SPLINE
SPL {X  -126.527, Y  +769.417, Z    +0.000, E1  +405.012, E3 -205837.853}
SPL {X  -145.458, Y  +738.125, Z    +0.000, E1  +396.959, E3 -205873.935}
SPL {X  -156.272, Y  +705.789, Z    +0.000, E1  +383.396, E3 -205888.344}
SPL {X  -159.413, Y  +685.076, Z    +0.000, E1  +371.341, E3 -205892.483}
SPL {X  -159.901, Y  +676.826, Z    +0.000, E1  +365.664, E3 -205893.315}
SPL {X  -159.990, Y  +671.106, Z    +0.000, E1  +361.459, E3 -205893.577}
SPL {X  -159.990, Y  +668.525, Z    +0.000, E1  +359.125, E3 -205893.622}
SPL {X  -159.990, Y  +664.817, Z    +0.000, E1  +353.836, E3 -205893.763}
SPL {X  -159.990, Y  +661.286, Z    +0.000, E1  +348.294, E3 -205894.024}
SPL {X  -159.990, Y  +654.198, Z    +0.000, E1  +336.753, E3 -205894.936}
SPL {X  -159.990, Y  +643.777, Z    +0.000, E1  +322.140, E3 -205897.101}
SPL {X  -159.990, Y  +634.027, Z    +0.000, E1  +313.116, E3 -205900.013}
SPL {X  -159.990, Y  +589.014, Z    +0.000, E1  +298.500, E3 -205920.064}
SPL {X  -159.990, Y  +484.717, Z    +0.000, E1  +295.169, E3 -205998.247}
SPL {X  -159.990, Y  +469.712, Z    +0.000, E1  +295.152, E3 -206013.185}
SPL {X  -159.990, Y  +456.089, Z    +0.000, E1  +295.174, E3 -206026.800}
SPL {X  -159.990, Y  +443.816, Z    +0.000, E1  +295.158, E3 -206039.000}
SPL {X  -159.990, Y  +405.035, Z    +0.000, E1  +292.209, E3 -206051.271}
SPL {X  -159.990, Y  +395.217, Z    +0.000, E1  +293.078, E3 -206067.380}
SPL {X  -159.990, Y  +385.177, Z    +0.000, E1  +294.011, E3 -206084.069}
SPL {X  -159.935, Y  +378.300, Z    +0.000, E1  +295.100, E3 -206099.278}
SPL {X  -159.533, Y  +370.414, Z    +0.000, E1  +296.253, E3 -206116.187}
SPL {X  -158.431, Y  +360.219, Z    +0.000, E1  +296.670, E3 -206129.704}
SPL {X  -157.299, Y  +353.279, Z    +0.000, E1  +296.835, E3 -206138.201}
SPL {X  -155.242, Y  +343.812, Z    +0.000, E1  +297.102, E3 -206150.249}
SPL {X  -151.999, Y  +332.569, Z    +0.000, E1  +297.592, E3 -206165.407}
SPL {X  -148.909, Y  +323.994, Z    +0.000, E1  +298.107, E3 -206177.581}
SPL {X  -146.667, Y  +318.581, Z    +0.000, E1  +298.485, E3 -206185.501}
SPL {X  -144.416, Y  +313.647, Z    +0.000, E1  +298.845, E3 -206192.837}
SPL {X  -141.484, Y  +307.808, Z    +0.000, E1  +299.342, E3 -206201.730}
SPL {X  -139.055, Y  +303.377, Z    +0.000, E1  +299.788, E3 -206208.642}
SPL {X  -136.464, Y  +298.988, Z    +0.000, E1  +300.231, E3 -206215.517}
SPL {X  -133.486, Y  +294.305, Z    +0.000, E1  +300.785, E3 -206222.979}
SPL {X  -111.198, Y  +267.470, Z    +0.000, E1  +308.990, E3 -206323.999}
ENDSPLINE

SPLINE
SPL {X  -136.508, Y  +299.059, Z    +0.000, E1  +318.212, E3 -206434.935}
SPL {X  -153.176, Y  +336.305, Z    +0.000, E1  +330.872, E3 -206461.500}
SPL {X  -158.263, Y  +359.056, Z    +0.000, E1  +342.551, E3 -206468.175}
SPL {X  -159.616, Y  +371.564, Z    +0.000, E1  +350.434, E3 -206470.080}
SPL {X  -159.983, Y  +381.031, Z    +0.000, E1  +357.053, E3 -206470.771}
SPL {X  -159.990, Y  +384.524, Z    +0.000, E1  +359.995, E3 -206470.859}
SPL {X  -159.990, Y  +386.890, Z    +0.000, E1  +362.742, E3 -206470.915}
SPL {X  -159.990, Y  +392.248, Z    +0.000, E1  +370.895, E3 -206471.242}
SPL {X  -159.990, Y  +398.030, Z    +0.000, E1  +380.706, E3 -206471.894}
SPL {X  -159.990, Y  +404.858, Z    +0.000, E1  +391.125, E3 -206473.138}
SPL {X  -159.990, Y  +416.328, Z    +0.000, E1  +404.105, E3 -206476.075}
SPL {X  -159.990, Y  +459.824, Z    +0.000, E1  +420.326, E3 -206495.997}
SPL {X  -159.990, Y  +561.459, Z    +0.000, E1  +423.923, E3 -206574.863}
SPL {X  -159.990, Y  +574.787, Z    +0.000, E1  +423.950, E3 -206588.660}
SPL {X  -159.990, Y  +590.041, Z    +0.000, E1  +423.939, E3 -206604.520}
SPL {X  -159.990, Y  +601.352, Z    +0.000, E1  +423.918, E3 -206616.306}
SPL {X  -159.990, Y  +610.973, Z    +0.000, E1  +423.927, E3 -206626.274}
SPL {X  -159.990, Y  +624.756, Z    +0.000, E1  +423.949, E3 -206640.552}
SPL {X  -159.990, Y  +640.674, Z    +0.000, E1  +423.943, E3 -206657.089}
SPL {X  -159.990, Y  +652.355, Z    +0.000, E1  +423.915, E3 -206669.287}
SPL {X  -159.990, Y  +661.195, Z    +0.000, E1  +423.915, E3 -206678.486}
SPL {X  -159.965, Y  +674.349, Z    +0.000, E1  +423.939, E3 -206692.123}
SPL {X  -159.404, Y  +685.179, Z    +0.000, E1  +423.831, E3 -206704.002}
SPL {X  -158.535, Y  +693.032, Z    +0.000, E1  +423.713, E3 -206713.051}
SPL {X  -156.949, Y  +702.544, Z    +0.000, E1  +423.501, E3 -206724.557}
SPL {X  -154.903, Y  +711.525, Z    +0.000, E1  +423.186, E3 -206736.028}
SPL {X  -153.138, Y  +717.820, Z    +0.000, E1  +422.909, E3 -206744.382}
SPL {X  -151.229, Y  +723.716, Z    +0.000, E1  +422.630, E3 -206752.392}
SPL {X  -148.422, Y  +731.231, Z    +0.000, E1  +422.207, E3 -206762.950}
SPL {X  -145.802, Y  +737.367, Z    +0.000, E1  +421.758, E3 -206771.902}
SPL {X  -143.476, Y  +742.291, Z    +0.000, E1  +421.379, E3 -206779.203}
SPL {X  -141.015, Y  +747.074, Z    +0.000, E1  +420.958, E3 -206786.459}
SPL {X  -138.539, Y  +751.523, Z    +0.000, E1  +420.526, E3 -206793.294}
SPL {X  -136.299, Y  +755.281, Z    +0.000, E1  +420.128, E3 -206799.155}
SPL {X  -133.306, Y  +759.967, Z    +0.000, E1  +419.584, E3 -206806.550}
SPL {X  -112.019, Y  +785.730, Z    +0.000, E1  +410.795, E3 -206909.290}
ENDSPLINE

SPLINE
SPL {X  -138.335, Y  +751.876, Z    +0.000, E1  +401.001, E3 -207023.589}
SPL {X  -153.384, Y  +716.997, Z    +0.000, E1  +388.774, E3 -207045.960}
SPL {X  -158.303, Y  +694.673, Z    +0.000, E1  +377.238, E3 -207052.272}
SPL {X  -159.604, Y  +682.609, Z    +0.000, E1  +369.664, E3 -207054.082}
SPL {X  -159.964, Y  +674.389, Z    +0.000, E1  +363.956, E3 -207054.744}
SPL {X  -159.990, Y  +669.409, Z    +0.000, E1  +360.015, E3 -207054.897}
SPL {X  -159.990, Y  +666.004, Z    +0.000, E1  +355.742, E3 -207054.998}
SPL {X  -159.990, Y  +661.286, Z    +0.000, E1  +348.294, E3 -207055.315}
SPL {X  -159.990, Y  +656.470, Z    +0.000, E1  +340.220, E3 -207055.852}
SPL {X  -159.990, Y  +651.555, Z    +0.000, E1  +332.416, E3 -207056.660}
SPL {X  -159.990, Y  +640.109, Z    +0.000, E1  +318.471, E3 -207059.489}
SPL {X  -159.990, Y  +589.014, Z    +0.000, E1  +298.500, E3 -207081.355}
SPL {X  -159.990, Y  +484.717, Z    +0.000, E1  +295.169, E3 -207159.538}
SPL {X  -159.990, Y  +474.300, Z    +0.000, E1  +295.184, E3 -207169.966}
SPL {X  -159.990, Y  +460.248, Z    +0.000, E1  +295.138, E3 -207183.876}
SPL {X  -159.990, Y  +443.816, Z    +0.000, E1  +295.158, E3 -207200.291}
SPL {X  -159.990, Y  +405.035, Z    +0.000, E1  +292.209, E3 -207212.562}
SPL {X  -159.990, Y  +397.824, Z    +0.000, E1  +292.709, E3 -207222.924}
SPL {X  -159.990, Y  +393.786, Z    +0.000, E1  +293.391, E3 -207232.243}
SPL {X  -159.990, Y  +387.038, Z    +0.000, E1  +293.844, E3 -207242.098}
SPL {X  -159.983, Y  +380.995, Z    +0.000, E1  +294.559, E3 -207253.667}
SPL {X  -159.898, Y  +377.064, Z    +0.000, E1  +295.481, E3 -207264.481}
SPL {X  -159.533, Y  +370.414, Z    +0.000, E1  +296.253, E3 -207277.478}
SPL {X  -158.431, Y  +360.219, Z    +0.000, E1  +296.670, E3 -207290.995}
SPL {X  -156.653, Y  +349.995, Z    +0.000, E1  +296.892, E3 -207303.563}
SPL {X  -153.792, Y  +338.401, Z    +0.000, E1  +297.323, E3 -207318.732}
SPL {X  -151.244, Y  +330.327, Z    +0.000, E1  +297.748, E3 -207329.885}
SPL {X  -148.909, Y  +323.994, Z    +0.000, E1  +298.107, E3 -207338.871}
SPL {X  -146.667, Y  +318.581, Z    +0.000, E1  +298.485, E3 -207346.791}
SPL {X  -144.416, Y  +313.647, Z    +0.000, E1  +298.845, E3 -207354.127}
SPL {X  -141.484, Y  +307.808, Z    +0.000, E1  +299.342, E3 -207363.020}
SPL {X  -139.055, Y  +303.377, Z    +0.000, E1  +299.788, E3 -207369.933}
SPL {X  -136.464, Y  +298.988, Z    +0.000, E1  +300.231, E3 -207376.807}
SPL {X  -133.486, Y  +294.305, Z    +0.000, E1  +300.785, E3 -207384.269}
SPL {X  -111.268, Y  +267.538, Z    +0.000, E1  +309.436, E3 -207492.168}
ENDSPLINE

SPLINE
SPL {X  -140.331, Y  +305.662, Z    +0.000, E1  +319.927, E3 -207604.236}
SPL {X  -153.176, Y  +336.305, Z    +0.000, E1  +330.872, E3 -207622.791}
SPL {X  -158.263, Y  +359.056, Z    +0.000, E1  +342.551, E3 -207629.465}
SPL {X  -159.616, Y  +371.564, Z    +0.000, E1  +350.434, E3 -207631.370}
SPL {X  -159.983, Y  +381.031, Z    +0.000, E1  +357.053, E3 -207632.061}
SPL {X  -159.990, Y  +384.524, Z    +0.000, E1  +359.995, E3 -207632.149}
SPL {X  -159.990, Y  +386.890, Z    +0.000, E1  +362.742, E3 -207632.205}
SPL {X  -159.990, Y  +392.248, Z    +0.000, E1  +370.895, E3 -207632.533}
SPL {X  -159.990, Y  +398.030, Z    +0.000, E1  +380.706, E3 -207633.184}
SPL {X  -159.990, Y  +404.858, Z    +0.000, E1  +391.125, E3 -207634.428}
SPL {X  -159.990, Y  +416.328, Z    +0.000, E1  +404.105, E3 -207637.365}
SPL {X  -159.990, Y  +459.824, Z    +0.000, E1  +420.326, E3 -207657.287}
SPL {X  -159.990, Y  +565.974, Z    +0.000, E1  +423.959, E3 -207740.776}
SPL {X  -159.990, Y  +582.903, Z    +0.000, E1  +423.951, E3 -207758.373}
SPL {X  -159.990, Y  +598.374, Z    +0.000, E1  +423.941, E3 -207774.459}
SPL {X  -159.990, Y  +614.998, Z    +0.000, E1  +423.962, E3 -207791.681}
SPL {X  -159.990, Y  +632.576, Z    +0.000, E1  +423.953, E3 -207809.947}
SPL {X  -159.990, Y  +648.849, Z    +0.000, E1  +423.945, E3 -207826.876}
SPL {X  -159.990, Y  +665.748, Z    +0.000, E1  +423.953, E3 -207844.431}
SPL {X  -159.643, Y  +682.032, Z    +0.000, E1  +423.894, E3 -207861.725}
SPL {X  -158.070, Y  +696.212, Z    +0.000, E1  +423.682, E3 -207878.063}
SPL {X  -155.481, Y  +709.215, Z    +0.000, E1  +423.310, E3 -207894.254}
SPL {X  -153.138, Y  +717.820, Z    +0.000, E1  +422.909, E3 -207905.672}
SPL {X  -151.229, Y  +723.716, Z    +0.000, E1  +422.630, E3 -207913.682}
SPL {X  -149.219, Y  +729.211, Z    +0.000, E1  +422.307, E3 -207921.390}
SPL {X  -146.537, Y  +735.716, Z    +0.000, E1  +421.906, E3 -207930.733}
SPL {X  -143.476, Y  +742.291, Z    +0.000, E1  +421.379, E3 -207940.493}
SPL {X  -141.015, Y  +747.074, Z    +0.000, E1  +420.958, E3 -207947.750}
SPL {X  -137.271, Y  +753.679, Z    +0.000, E1  +420.346, E3 -207957.888}
SPL {X  -133.306, Y  +759.967, Z    +0.000, E1  +419.584, E3 -207967.840}
SPL {X  -112.019, Y  +785.730, Z    +0.000, E1  +410.795, E3 -208070.581}
ENDSPLINE

SPLINE
SPL {X  -138.335, Y  +751.876, Z    +0.000, E1  +401.001, E3 -208184.879}
SPL {X  -150.285, Y  +726.376, Z    +0.000, E1  +392.667, E3 -208203.288}
SPL {X  -156.272, Y  +705.789, Z    +0.000, E1  +383.396, E3 -208210.925}
SPL {X  -159.413, Y  +685.076, Z    +0.000, E1  +371.341, E3 -208215.063}
SPL {X  -159.964, Y  +674.389, Z    +0.000, E1  +363.956, E3 -208216.034}
SPL {X  -159.990, Y  +670.214, Z    +0.000, E1  +360.653, E3 -208216.180}
SPL {X  -159.990, Y  +669.154, Z    +0.000, E1  +359.694, E3 -208216.189}
SPL {X  -159.990, Y  +666.004, Z    +0.000, E1  +355.742, E3 -208216.289}
SPL {X  -159.990, Y  +661.286, Z    +0.000, E1  +348.294, E3 -208216.605}
SPL {X  -159.990, Y  +656.470, Z    +0.000, E1  +340.220, E3 -208217.143}
SPL {X  -159.990, Y  +651.555, Z    +0.000, E1  +332.416, E3 -208217.950}
SPL {X  -159.990, Y  +640.109, Z    +0.000, E1  +318.471, E3 -208220.779}
SPL {X  -159.990, Y  +589.014, Z    +0.000, E1  +298.500, E3 -208242.645}
SPL {X  -159.990, Y  +484.717, Z    +0.000, E1  +295.169, E3 -208320.828}
SPL {X  -159.990, Y  +469.712, Z    +0.000, E1  +295.152, E3 -208335.765}
SPL {X  -159.990, Y  +456.089, Z    +0.000, E1  +295.174, E3 -208349.381}
SPL {X  -159.990, Y  +443.816, Z    +0.000, E1  +295.158, E3 -208361.581}
SPL {X  -159.990, Y  +405.035, Z    +0.000, E1  +292.209, E3 -208373.852}
SPL {X  -159.990, Y  +397.824, Z    +0.000, E1  +292.709, E3 -208384.214}
SPL {X  -159.990, Y  +393.786, Z    +0.000, E1  +293.391, E3 -208393.533}
SPL {X  -159.990, Y  +385.177, Z    +0.000, E1  +294.011, E3 -208406.649}
SPL {X  -159.935, Y  +378.300, Z    +0.000, E1  +295.100, E3 -208421.859}
SPL {X  -159.716, Y  +373.142, Z    +0.000, E1  +296.084, E3 -208434.400}
SPL {X  -158.852, Y  +363.449, Z    +0.000, E1  +296.568, E3 -208448.350}
SPL {X  -157.299, Y  +353.279, Z    +0.000, E1  +296.835, E3 -208460.782}
SPL {X  -155.242, Y  +343.812, Z    +0.000, E1  +297.102, E3 -208472.830}
SPL {X  -151.999, Y  +332.569, Z    +0.000, E1  +297.592, E3 -208487.988}
SPL {X  -148.909, Y  +323.994, Z    +0.000, E1  +298.107, E3 -208500.161}
SPL {X  -146.667, Y  +318.581, Z    +0.000, E1  +298.485, E3 -208508.082}
SPL {X  -144.416, Y  +313.647, Z    +0.000, E1  +298.845, E3 -208515.418}
SPL {X  -141.484, Y  +307.808, Z    +0.000, E1  +299.342, E3 -208524.311}
SPL {X  -139.055, Y  +303.377, Z    +0.000, E1  +299.788, E3 -208531.223}
SPL {X  -136.464, Y  +298.988, Z    +0.000, E1  +300.231, E3 -208538.097}
SPL {X  -133.486, Y  +294.305, Z    +0.000, E1  +300.785, E3 -208545.560}
SPL {X  -111.268, Y  +267.538, Z    +0.000, E1  +309.436, E3 -208653.459}
ENDSPLINE

SPLINE
SPL {X  -140.331, Y  +305.662, Z    +0.000, E1  +319.927, E3 -208765.527}
SPL {X  -153.176, Y  +336.305, Z    +0.000, E1  +330.872, E3 -208784.081}
SPL {X  -158.263, Y  +359.056, Z    +0.000, E1  +342.551, E3 -208790.756}
SPL {X  -159.616, Y  +371.564, Z    +0.000, E1  +350.434, E3 -208792.661}
SPL {X  -159.946, Y  +378.747, Z    +0.000, E1  +355.440, E3 -208793.256}
SPL {X  -159.990, Y  +384.172, Z    +0.000, E1  +359.586, E3 -208793.434}
SPL {X  -159.990, Y  +385.853, Z    +0.000, E1  +361.539, E3 -208793.459}
SPL {X  -159.990, Y  +389.234, Z    +0.000, E1  +366.142, E3 -208793.604}
SPL {X  -159.990, Y  +395.814, Z    +0.000, E1  +376.762, E3 -208794.205}
SPL {X  -159.990, Y  +404.858, Z    +0.000, E1  +391.125, E3 -208795.718}
SPL {X  -159.990, Y  +416.328, Z    +0.000, E1  +404.105, E3 -208798.655}
SPL {X  -159.990, Y  +459.824, Z    +0.000, E1  +420.326, E3 -208818.577}
SPL {X  -159.990, Y  +565.974, Z    +0.000, E1  +423.959, E3 -208902.066}
SPL {X  -159.990, Y  +578.588, Z    +0.000, E1  +423.918, E3 -208915.245}
SPL {X  -159.990, Y  +590.041, Z    +0.000, E1  +423.939, E3 -208927.100}
SPL {X  -159.990, Y  +601.352, Z    +0.000, E1  +423.918, E3 -208938.887}
SPL {X  -159.990, Y  +610.973, Z    +0.000, E1  +423.927, E3 -208948.855}
SPL {X  -159.990, Y  +624.756, Z    +0.000, E1  +423.949, E3 -208963.133}
SPL {X  -159.990, Y  +636.914, Z    +0.000, E1  +423.917, E3 -208975.808}
SPL {X  -159.990, Y  +648.849, Z    +0.000, E1  +423.945, E3 -208988.166}
SPL {X  -159.990, Y  +661.195, Z    +0.000, E1  +423.915, E3 -209001.067}
SPL {X  -159.965, Y  +674.349, Z    +0.000, E1  +423.939, E3 -209014.703}
SPL {X  -159.404, Y  +685.179, Z    +0.000, E1  +423.831, E3 -209026.582}
SPL {X  -158.535, Y  +693.032, Z    +0.000, E1  +423.713, E3 -209035.632}
SPL {X  -156.949, Y  +702.544, Z    +0.000, E1  +423.501, E3 -209047.137}
SPL {X  -154.903, Y  +711.525, Z    +0.000, E1  +423.186, E3 -209058.608}
SPL {X  -153.138, Y  +717.820, Z    +0.000, E1  +422.909, E3 -209066.963}
SPL {X  -151.229, Y  +723.716, Z    +0.000, E1  +422.630, E3 -209074.972}
SPL {X  -149.219, Y  +729.211, Z    +0.000, E1  +422.307, E3 -209082.681}
SPL {X  -146.537, Y  +735.716, Z    +0.000, E1  +421.906, E3 -209092.024}
SPL {X  -143.476, Y  +742.291, Z    +0.000, E1  +421.379, E3 -209101.784}
SPL {X  -141.015, Y  +747.074, Z    +0.000, E1  +420.958, E3 -209109.040}
SPL {X  -137.271, Y  +753.679, Z    +0.000, E1  +420.346, E3 -209119.179}
SPL {X  -133.306, Y  +759.967, Z    +0.000, E1  +419.584, E3 -209129.130}
SPL {X  -112.019, Y  +785.730, Z    +0.000, E1  +410.795, E3 -209231.871}
ENDSPLINE

SPLINE
SPL {X  -138.335, Y  +751.876, Z    +0.000, E1  +401.001, E3 -209346.170}
SPL {X  -150.285, Y  +726.376, Z    +0.000, E1  +392.667, E3 -209364.579}
SPL {X  -156.272, Y  +705.789, Z    +0.000, E1  +383.396, E3 -209372.215}
SPL {X  -159.413, Y  +685.076, Z    +0.000, E1  +371.341, E3 -209376.354}
SPL {X  -159.964, Y  +674.389, Z    +0.000, E1  +363.956, E3 -209377.324}
SPL {X  -159.990, Y  +669.409, Z    +0.000, E1  +360.015, E3 -209377.477}
SPL {X  -159.990, Y  +667.272, Z    +0.000, E1  +357.329, E3 -209377.521}
SPL {X  -159.990, Y  +664.817, Z    +0.000, E1  +353.836, E3 -209377.634}
SPL {X  -159.990, Y  +661.286, Z    +0.000, E1  +348.294, E3 -209377.895}
SPL {X  -159.990, Y  +654.198, Z    +0.000, E1  +336.753, E3 -209378.807}
SPL {X  -159.990, Y  +640.109, Z    +0.000, E1  +318.471, E3 -209382.070}
SPL {X  -159.990, Y  +589.014, Z    +0.000, E1  +298.500, E3 -209403.935}
SPL {X  -159.990, Y  +484.717, Z    +0.000, E1  +295.169, E3 -209482.118}
SPL {X  -159.990, Y  +474.300, Z    +0.000, E1  +295.184, E3 -209492.546}
SPL {X  -159.990, Y  +465.825, Z    +0.000, E1  +295.182, E3 -209500.986}
SPL {X  -159.990, Y  +451.559, Z    +0.000, E1  +295.138, E3 -209515.123}
SPL {X  -159.990, Y  +438.393, Z    +0.000, E1  +295.184, E3 -209528.344}
SPL {X  -159.990, Y  +405.035, Z    +0.000, E1  +292.209, E3 -209535.142}
SPL {X  -159.990, Y  +395.217, Z    +0.000, E1  +293.078, E3 -209551.251}
SPL {X  -159.990, Y  +387.038, Z    +0.000, E1  +293.844, E3 -209564.679}
SPL {X  -159.983, Y  +380.995, Z    +0.000, E1  +294.559, E3 -209576.248}
SPL {X  -159.795, Y  +374.602, Z    +0.000, E1  +295.796, E3 -209592.267}
SPL {X  -158.852, Y  +363.449, Z    +0.000, E1  +296.568, E3 -209609.640}
SPL {X  -156.653, Y  +349.995, Z    +0.000, E1  +296.892, E3 -209626.144}
SPL {X  -153.792, Y  +338.401, Z    +0.000, E1  +297.323, E3 -209641.313}
SPL {X  -151.244, Y  +330.327, Z    +0.000, E1  +297.748, E3 -209652.466}
SPL {X  -148.909, Y  +323.994, Z    +0.000, E1  +298.107, E3 -209661.452}
SPL {X  -146.667, Y  +318.581, Z    +0.000, E1  +298.485, E3 -209669.372}
SPL {X  -144.416, Y  +313.647, Z    +0.000, E1  +298.845, E3 -209676.708}
SPL {X  -141.484, Y  +307.808, Z    +0.000, E1  +299.342, E3 -209685.601}
SPL {X  -139.055, Y  +303.377, Z    +0.000, E1  +299.788, E3 -209692.513}
SPL {X  -136.464, Y  +298.988, Z    +0.000, E1  +300.231, E3 -209699.388}
SPL {X  -133.486, Y  +294.305, Z    +0.000, E1  +300.785, E3 -209706.850}
SPL {X  -111.268, Y  +267.538, Z    +0.000, E1  +309.436, E3 -209814.749}
ENDSPLINE

SPLINE
SPL {X  -140.331, Y  +305.662, Z    +0.000, E1  +319.927, E3 -209926.817}
SPL {X  -153.176, Y  +336.305, Z    +0.000, E1  +330.872, E3 -209945.371}
SPL {X  -157.724, Y  +355.668, Z    +0.000, E1  +340.639, E3 -209951.379}
SPL {X  -159.465, Y  +369.545, Z    +0.000, E1  +349.053, E3 -209953.702}
SPL {X  -159.983, Y  +381.031, Z    +0.000, E1  +357.053, E3 -209954.642}
SPL {X  -159.990, Y  +384.524, Z    +0.000, E1  +359.995, E3 -209954.730}
SPL {X  -159.990, Y  +386.890, Z    +0.000, E1  +362.742, E3 -209954.786}
SPL {X  -159.990, Y  +392.248, Z    +0.000, E1  +370.895, E3 -209955.113}
SPL {X  -159.990, Y  +398.030, Z    +0.000, E1  +380.706, E3 -209955.765}
SPL {X  -159.990, Y  +404.858, Z    +0.000, E1  +391.125, E3 -209957.009}
SPL {X  -159.990, Y  +416.328, Z    +0.000, E1  +404.105, E3 -209959.946}
SPL {X  -159.990, Y  +459.824, Z    +0.000, E1  +420.326, E3 -209979.868}
SPL {X  -159.990, Y  +565.974, Z    +0.000, E1  +423.959, E3 -210063.357}
SPL {X  -159.990, Y  +578.588, Z    +0.000, E1  +423.918, E3 -210076.536}
SPL {X  -159.990, Y  +590.041, Z    +0.000, E1  +423.939, E3 -210088.391}
SPL {X  -159.990, Y  +601.352, Z    +0.000, E1  +423.918, E3 -210100.177}
SPL {X  -159.990, Y  +614.998, Z    +0.000, E1  +423.962, E3 -210114.262}
SPL {X  -159.990, Y  +628.256, Z    +0.000, E1  +423.919, E3 -210128.110}
SPL {X  -159.990, Y  +640.674, Z    +0.000, E1  +423.943, E3 -210140.960}
SPL {X  -159.990, Y  +657.298, Z    +0.000, E1  +423.953, E3 -210158.232}
SPL {X  -159.990, Y  +670.369, Z    +0.000, E1  +423.912, E3 -210171.889}
SPL {X  -159.643, Y  +682.032, Z    +0.000, E1  +423.894, E3 -210184.305}
SPL {X  -158.070, Y  +696.212, Z    +0.000, E1  +423.682, E3 -210200.643}
SPL {X  -155.481, Y  +709.215, Z    +0.000, E1  +423.310, E3 -210216.834}
SPL {X  -153.138, Y  +717.820, Z    +0.000, E1  +422.909, E3 -210228.253}
SPL {X  -151.229, Y  +723.716, Z    +0.000, E1  +422.630, E3 -210236.263}
SPL {X  -149.219, Y  +729.211, Z    +0.000, E1  +422.307, E3 -210243.971}
SPL {X  -146.537, Y  +735.716, Z    +0.000, E1  +421.906, E3 -210253.314}
SPL {X  -143.476, Y  +742.291, Z    +0.000, E1  +421.379, E3 -210263.074}
SPL {X  -141.015, Y  +747.074, Z    +0.000, E1  +420.958, E3 -210270.330}
SPL {X  -137.271, Y  +753.679, Z    +0.000, E1  +420.346, E3 -210280.469}
SPL {X  -133.306, Y  +759.967, Z    +0.000, E1  +419.584, E3 -210290.421}
SPL {X  -112.019, Y  +785.730, Z    +0.000, E1  +410.795, E3 -210393.161}
ENDSPLINE

SPLINE
SPL {X  -126.527, Y  +769.417, Z    +0.000, E1  +405.012, E3 -210483.014}
SPL {X  -141.954, Y  +745.296, Z    +0.000, E1  +399.179, E3 -210514.212}
SPL {X  -153.384, Y  +716.997, Z    +0.000, E1  +388.774, E3 -210529.831}
SPL {X  -158.303, Y  +694.673, Z    +0.000, E1  +377.238, E3 -210536.143}
SPL {X  -159.604, Y  +682.609, Z    +0.000, E1  +369.664, E3 -210537.953}
SPL {X  -159.964, Y  +674.389, Z    +0.000, E1  +363.956, E3 -210538.614}
SPL {X  -159.990, Y  +669.409, Z    +0.000, E1  +360.015, E3 -210538.768}
SPL {X  -159.990, Y  +666.004, Z    +0.000, E1  +355.742, E3 -210538.869}
SPL {X  -159.990, Y  +661.286, Z    +0.000, E1  +348.294, E3 -210539.186}
SPL {X  -159.990, Y  +654.198, Z    +0.000, E1  +336.753, E3 -210540.097}
SPL {X  -159.990, Y  +640.109, Z    +0.000, E1  +318.471, E3 -210543.360}
SPL {X  -159.990, Y  +589.014, Z    +0.000, E1  +298.500, E3 -210565.226}
SPL {X  -159.990, Y  +484.717, Z    +0.000, E1  +295.169, E3 -210643.409}
SPL {X  -159.990, Y  +474.300, Z    +0.000, E1  +295.184, E3 -210653.836}
SPL {X  -159.990, Y  +465.825, Z    +0.000, E1  +295.182, E3 -210662.276}
SPL {X  -159.990, Y  +451.559, Z    +0.000, E1  +295.138, E3 -210676.413}
SPL {X  -159.990, Y  +423.512, Z    +0.000, E1  +293.559, E3 -210690.847}
SPL {X  -159.990, Y  +399.563, Z    +0.000, E1  +292.427, E3 -210703.125}
SPL {X  -159.990, Y  +393.786, Z    +0.000, E1  +293.391, E3 -210716.113}
SPL {X  -159.990, Y  +387.038, Z    +0.000, E1  +293.844, E3 -210725.969}
SPL {X  -159.983, Y  +380.995, Z    +0.000, E1  +294.559, E3 -210737.538}
SPL {X  -159.898, Y  +377.064, Z    +0.000, E1  +295.481, E3 -210748.352}
SPL {X  -159.716, Y  +373.142, Z    +0.000, E1  +296.084, E3 -210756.980}
SPL {X  -158.852, Y  +363.449, Z    +0.000, E1  +296.568, E3 -210770.930}
SPL {X  -157.299, Y  +353.279, Z    +0.000, E1  +296.835, E3 -210783.362}
SPL {X  -155.242, Y  +343.812, Z    +0.000, E1  +297.102, E3 -210795.410}
SPL {X  -151.999, Y  +332.569, Z    +0.000, E1  +297.592, E3 -210810.568}
SPL {X  -148.909, Y  +323.994, Z    +0.000, E1  +298.107, E3 -210822.742}
SPL {X  -146.667, Y  +318.581, Z    +0.000, E1  +298.485, E3 -210830.662}
SPL {X  -144.416, Y  +313.647, Z    +0.000, E1  +298.845, E3 -210837.998}
SPL {X  -141.484, Y  +307.808, Z    +0.000, E1  +299.342, E3 -210846.891}
SPL {X  -139.055, Y  +303.377, Z    +0.000, E1  +299.788, E3 -210853.804}
SPL {X  -136.464, Y  +298.988, Z    +0.000, E1  +300.231, E3 -210860.678}
SPL {X  -133.486, Y  +294.305, Z    +0.000, E1  +300.785, E3 -210868.140}
SPL {X  -111.268, Y  +267.538, Z    +0.000, E1  +309.436, E3 -210976.039}
ENDSPLINE

SPLINE
SPL {X  -140.331, Y  +305.662, Z    +0.000, E1  +319.927, E3 -211088.107}
SPL {X  -153.176, Y  +336.305, Z    +0.000, E1  +330.872, E3 -211106.662}
SPL {X  -158.263, Y  +359.056, Z    +0.000, E1  +342.551, E3 -211113.336}
SPL {X  -159.616, Y  +371.564, Z    +0.000, E1  +350.434, E3 -211115.241}
SPL {X  -159.983, Y  +381.031, Z    +0.000, E1  +357.053, E3 -211115.932}
SPL {X  -159.990, Y  +385.049, Z    +0.000, E1  +360.437, E3 -211116.028}
SPL {X  -159.990, Y  +389.234, Z    +0.000, E1  +366.142, E3 -211116.184}
SPL {X  -159.990, Y  +395.814, Z    +0.000, E1  +376.762, E3 -211116.785}
SPL {X  -159.990, Y  +404.858, Z    +0.000, E1  +391.125, E3 -211118.299}
SPL {X  -159.990, Y  +416.328, Z    +0.000, E1  +404.105, E3 -211121.236}
SPL {X  -159.990, Y  +459.824, Z    +0.000, E1  +420.326, E3 -211141.158}
SPL {X  -159.990, Y  +565.974, Z    +0.000, E1  +423.959, E3 -211224.647}
SPL {X  -159.990, Y  +578.588, Z    +0.000, E1  +423.918, E3 -211237.826}
SPL {X  -159.990, Y  +590.041, Z    +0.000, E1  +423.939, E3 -211249.681}
SPL {X  -159.990, Y  +601.352, Z    +0.000, E1  +423.918, E3 -211261.467}
SPL {X  -159.990, Y  +610.973, Z    +0.000, E1  +423.927, E3 -211271.436}
SPL {X  -159.990, Y  +624.756, Z    +0.000, E1  +423.949, E3 -211285.713}
SPL {X  -159.990, Y  +640.674, Z    +0.000, E1  +423.943, E3 -211302.250}
SPL {X  -159.990, Y  +657.298, Z    +0.000, E1  +423.953, E3 -211319.522}
SPL {X  -159.965, Y  +674.349, Z    +0.000, E1  +423.939, E3 -211337.284}
SPL {X  -159.404, Y  +685.179, Z    +0.000, E1  +423.831, E3 -211349.163}
SPL {X  -158.535, Y  +693.032, Z    +0.000, E1  +423.713, E3 -211358.213}
SPL {X  -156.949, Y  +702.544, Z    +0.000, E1  +423.501, E3 -211369.718}
SPL {X  -154.903, Y  +711.525, Z    +0.000, E1  +423.186, E3 -211381.189}
SPL {X  -153.138, Y  +717.820, Z    +0.000, E1  +422.909, E3 -211389.543}
SPL {X  -151.229, Y  +723.716, Z    +0.000, E1  +422.630, E3 -211397.553}
SPL {X  -149.219, Y  +729.211, Z    +0.000, E1  +422.307, E3 -211405.261}
SPL {X  -146.537, Y  +735.716, Z    +0.000, E1  +421.906, E3 -211414.604}
SPL {X  -143.476, Y  +742.291, Z    +0.000, E1  +421.379, E3 -211424.364}
SPL {X  -141.015, Y  +747.074, Z    +0.000, E1  +420.958, E3 -211431.621}
SPL {X  -138.539, Y  +751.523, Z    +0.000, E1  +420.526, E3 -211438.456}
SPL {X  -136.299, Y  +755.281, Z    +0.000, E1  +420.128, E3 -211444.317}
SPL {X  -133.306, Y  +759.967, Z    +0.000, E1  +419.584, E3 -211451.711}
SPL {X  -112.019, Y  +785.730, Z    +0.000, E1  +410.795, E3 -211554.452}
ENDSPLINE

SPLINE
SPL {X  -138.335, Y  +751.876, Z    +0.000, E1  +401.001, E3 -211668.750}
SPL {X  -153.384, Y  +716.997, Z    +0.000, E1  +388.774, E3 -211691.122}
SPL {X  -157.578, Y  +699.176, Z    +0.000, E1  +379.774, E3 -211696.551}
SPL {X  -159.413, Y  +685.076, Z    +0.000, E1  +371.341, E3 -211698.934}
SPL {X  -159.901, Y  +676.826, Z    +0.000, E1  +365.664, E3 -211699.767}
SPL {X  -159.990, Y  +671.106, Z    +0.000, E1  +361.459, E3 -211700.028}
SPL {X  -159.990, Y  +669.154, Z    +0.000, E1  +359.694, E3 -211700.060}
SPL {X  -159.990, Y  +666.004, Z    +0.000, E1  +355.742, E3 -211700.160}
SPL {X  -159.990, Y  +661.286, Z    +0.000, E1  +348.294, E3 -211700.476}
SPL {X  -159.990, Y  +654.198, Z    +0.000, E1  +336.753, E3 -211701.387}
SPL {X  -159.990, Y  +640.109, Z    +0.000, E1  +318.471, E3 -211704.650}
SPL {X  -159.990, Y  +589.014, Z    +0.000, E1  +298.500, E3 -211726.516}
SPL {X  -159.990, Y  +484.717, Z    +0.000, E1  +295.169, E3 -211804.699}
SPL {X  -159.990, Y  +469.712, Z    +0.000, E1  +295.152, E3 -211819.636}
SPL {X  -159.990, Y  +451.559, Z    +0.000, E1  +295.138, E3 -211837.703}
SPL {X  -159.990, Y  +423.512, Z    +0.000, E1  +293.559, E3 -211852.137}
SPL {X  -159.990, Y  +399.563, Z    +0.000, E1  +292.427, E3 -211864.415}
SPL {X  -159.990, Y  +393.786, Z    +0.000, E1  +293.391, E3 -211877.404}
SPL {X  -159.990, Y  +387.038, Z    +0.000, E1  +293.844, E3 -211887.260}
SPL {X  -159.983, Y  +380.995, Z    +0.000, E1  +294.559, E3 -211898.828}
SPL {X  -159.795, Y  +374.602, Z    +0.000, E1  +295.796, E3 -211914.848}
SPL {X  -159.306, Y  +367.719, Z    +0.000, E1  +296.544, E3 -211927.305}
SPL {X  -158.431, Y  +360.219, Z    +0.000, E1  +296.670, E3 -211936.156}
SPL {X  -157.299, Y  +353.279, Z    +0.000, E1  +296.835, E3 -211944.652}
SPL {X  -155.242, Y  +343.812, Z    +0.000, E1  +297.102, E3 -211956.701}
SPL {X  -151.999, Y  +332.569, Z    +0.000, E1  +297.592, E3 -211971.859}
SPL {X  -148.909, Y  +323.994, Z    +0.000, E1  +298.107, E3 -211984.032}
SPL {X  -146.667, Y  +318.581, Z    +0.000, E1  +298.485, E3 -211991.952}
SPL {X  -144.416, Y  +313.647, Z    +0.000, E1  +298.845, E3 -211999.289}
SPL {X  -141.484, Y  +307.808, Z    +0.000, E1  +299.342, E3 -212008.182}
SPL {X  -139.055, Y  +303.377, Z    +0.000, E1  +299.788, E3 -212015.094}
SPL {X  -136.464, Y  +298.988, Z    +0.000, E1  +300.231, E3 -212021.968}
SPL {X  -133.486, Y  +294.305, Z    +0.000, E1  +300.785, E3 -212029.431}
SPL {X  -111.268, Y  +267.538, Z    +0.000, E1  +309.436, E3 -212137.329}
ENDSPLINE

SPLINE
SPL {X  -140.331, Y  +305.662, Z    +0.000, E1  +319.927, E3 -212249.398}
SPL {X  -153.176, Y  +336.305, Z    +0.000, E1  +330.872, E3 -212267.952}
SPL {X  -157.724, Y  +355.668, Z    +0.000, E1  +340.639, E3 -212273.960}
SPL {X  -159.465, Y  +369.545, Z    +0.000, E1  +349.053, E3 -212276.283}
SPL {X  -159.983, Y  +381.031, Z    +0.000, E1  +357.053, E3 -212277.222}
SPL {X  -159.990, Y  +384.524, Z    +0.000, E1  +359.995, E3 -212277.310}
SPL {X  -159.990, Y  +386.890, Z    +0.000, E1  +362.742, E3 -212277.366}
SPL {X  -159.990, Y  +392.248, Z    +0.000, E1  +370.895, E3 -212277.694}
SPL {X  -159.990, Y  +398.030, Z    +0.000, E1  +380.706, E3 -212278.345}
SPL {X  -159.990, Y  +404.858, Z    +0.000, E1  +391.125, E3 -212279.589}
SPL {X  -159.990, Y  +416.328, Z    +0.000, E1  +404.105, E3 -212282.526}
SPL {X  -159.990, Y  +459.824, Z    +0.000, E1  +420.326, E3 -212302.448}
SPL {X  -159.990, Y  +561.459, Z    +0.000, E1  +423.923, E3 -212381.315}
SPL {X  -159.990, Y  +574.787, Z    +0.000, E1  +423.950, E3 -212395.111}
SPL {X  -159.990, Y  +590.041, Z    +0.000, E1  +423.939, E3 -212410.971}
SPL {X  -159.990, Y  +601.352, Z    +0.000, E1  +423.918, E3 -212422.758}
SPL {X  -159.990, Y  +610.973, Z    +0.000, E1  +423.927, E3 -212432.726}
SPL {X  -159.990, Y  +624.756, Z    +0.000, E1  +423.949, E3 -212447.004}
SPL {X  -159.990, Y  +640.674, Z    +0.000, E1  +423.943, E3 -212463.540}
SPL {X  -159.990, Y  +652.355, Z    +0.000, E1  +423.915, E3 -212475.739}
SPL {X  -159.990, Y  +661.195, Z    +0.000, E1  +423.915, E3 -212484.938}
SPL {X  -159.965, Y  +674.349, Z    +0.000, E1  +423.939, E3 -212498.574}
SPL {X  -159.404, Y  +685.179, Z    +0.000, E1  +423.831, E3 -212510.453}
SPL {X  -158.535, Y  +693.032, Z    +0.000, E1  +423.713, E3 -212519.503}
SPL {X  -156.949, Y  +702.544, Z    +0.000, E1  +423.501, E3 -212531.008}
SPL {X  -154.903, Y  +711.525, Z    +0.000, E1  +423.186, E3 -212542.479}
SPL {X  -153.138, Y  +717.820, Z    +0.000, E1  +422.909, E3 -212550.834}
SPL {X  -151.229, Y  +723.716, Z    +0.000, E1  +422.630, E3 -212558.843}
SPL {X  -149.219, Y  +729.211, Z    +0.000, E1  +422.307, E3 -212566.552}
SPL {X  -146.537, Y  +735.716, Z    +0.000, E1  +421.906, E3 -212575.895}
SPL {X  -143.476, Y  +742.291, Z    +0.000, E1  +421.379, E3 -212585.655}
SPL {X  -141.015, Y  +747.074, Z    +0.000, E1  +420.958, E3 -212592.911}
SPL {X  -138.539, Y  +751.523, Z    +0.000, E1  +420.526, E3 -212599.746}
SPL {X  -136.299, Y  +755.281, Z    +0.000, E1  +420.128, E3 -212605.607}
SPL {X  -133.306, Y  +759.967, Z    +0.000, E1  +419.584, E3 -212613.001}
SPL {X  -112.019, Y  +785.730, Z    +0.000, E1  +410.795, E3 -212715.742}
ENDSPLINE

SPLINE
SPL {X  -126.527, Y  +769.417, Z    +0.000, E1  +405.012, E3 -212805.594}
SPL {X  -145.458, Y  +738.125, Z    +0.000, E1  +396.959, E3 -212841.677}
SPL {X  -156.272, Y  +705.789, Z    +0.000, E1  +383.396, E3 -212856.086}
SPL {X  -159.413, Y  +685.076, Z    +0.000, E1  +371.341, E3 -212860.225}
SPL {X  -159.901, Y  +676.826, Z    +0.000, E1  +365.664, E3 -212861.057}
SPL {X  -159.990, Y  +671.106, Z    +0.000, E1  +361.459, E3 -212861.319}
SPL {X  -159.990, Y  +668.525, Z    +0.000, E1  +359.125, E3 -212861.364}
SPL {X  -159.990, Y  +664.817, Z    +0.000, E1  +353.836, E3 -212861.505}
SPL {X  -159.990, Y  +661.286, Z    +0.000, E1  +348.294, E3 -212861.766}
SPL {X  -159.990, Y  +654.198, Z    +0.000, E1  +336.753, E3 -212862.678}
SPL {X  -159.990, Y  +643.777, Z    +0.000, E1  +322.140, E3 -212864.843}
SPL {X  -159.990, Y  +634.027, Z    +0.000, E1  +313.116, E3 -212867.755}
SPL {X  -159.990, Y  +589.014, Z    +0.000, E1  +298.500, E3 -212887.806}
SPL {X  -159.990, Y  +484.717, Z    +0.000, E1  +295.169, E3 -212965.989}
SPL {X  -159.990, Y  +469.712, Z    +0.000, E1  +295.152, E3 -212980.926}
SPL {X  -159.990, Y  +456.089, Z    +0.000, E1  +295.174, E3 -212994.542}
SPL {X  -159.990, Y  +443.816, Z    +0.000, E1  +295.158, E3 -213006.742}
SPL {X  -159.990, Y  +405.035, Z    +0.000, E1  +292.209, E3 -213019.013}
SPL {X  -159.990, Y  +395.217, Z    +0.000, E1  +293.078, E3 -213035.122}
SPL {X  -159.990, Y  +385.177, Z    +0.000, E1  +294.011, E3 -213051.811}
SPL {X  -159.935, Y  +378.300, Z    +0.000, E1  +295.100, E3 -213067.020}
SPL {X  -159.533, Y  +370.414, Z    +0.000, E1  +296.253, E3 -213083.929}
SPL {X  -158.431, Y  +360.219, Z    +0.000, E1  +296.670, E3 -213097.446}
SPL {X  -157.299, Y  +353.279, Z    +0.000, E1  +296.835, E3 -213105.943}
SPL {X  -155.242, Y  +343.812, Z    +0.000, E1  +297.102, E3 -213117.991}
SPL {X  -151.999, Y  +332.569, Z    +0.000, E1  +297.592, E3 -213133.149}
SPL {X  -148.909, Y  +323.994, Z    +0.000, E1  +298.107, E3 -213145.322}
SPL {X  -146.667, Y  +318.581, Z    +0.000, E1  +298.485, E3 -213153.243}
SPL {X  -144.416, Y  +313.647, Z    +0.000, E1  +298.845, E3 -213160.579}
SPL {X  -141.484, Y  +307.808, Z    +0.000, E1  +299.342, E3 -213169.472}
SPL {X  -139.055, Y  +303.377, Z    +0.000, E1  +299.788, E3 -213176.384}
SPL {X  -136.464, Y  +298.988, Z    +0.000, E1  +300.231, E3 -213183.259}
SPL {X  -133.486, Y  +294.305, Z    +0.000, E1  +300.785, E3 -213190.721}
SPL {X  -111.198, Y  +267.470, Z    +0.000, E1  +308.990, E3 -213291.741}
ENDSPLINE

SPLINE
SPL {X  -136.508, Y  +299.059, Z    +0.000, E1  +318.212, E3 -213402.677}
SPL {X  -153.176, Y  +336.305, Z    +0.000, E1  +330.872, E3 -213429.242}
SPL {X  -158.263, Y  +359.056, Z    +0.000, E1  +342.551, E3 -213435.917}
SPL {X  -159.616, Y  +371.564, Z    +0.000, E1  +350.434, E3 -213437.822}
SPL {X  -159.983, Y  +381.031, Z    +0.000, E1  +357.053, E3 -213438.513}
SPL {X  -159.990, Y  +384.524, Z    +0.000, E1  +359.995, E3 -213438.601}
SPL {X  -159.990, Y  +386.890, Z    +0.000, E1  +362.742, E3 -213438.657}
SPL {X  -159.990, Y  +392.248, Z    +0.000, E1  +370.895, E3 -213438.984}
SPL {X  -159.990, Y  +398.030, Z    +0.000, E1  +380.706, E3 -213439.636}
SPL {X  -159.990, Y  +404.858, Z    +0.000, E1  +391.125, E3 -213440.880}
SPL {X  -159.990, Y  +416.328, Z    +0.000, E1  +404.105, E3 -213443.817}
SPL {X  -159.990, Y  +459.824, Z    +0.000, E1  +420.326, E3 -213463.739}
SPL {X  -159.990, Y  +561.459, Z    +0.000, E1  +423.923, E3 -213542.605}
SPL {X  -159.990, Y  +574.787, Z    +0.000, E1  +423.950, E3 -213556.402}
SPL {X  -159.990, Y  +590.041, Z    +0.000, E1  +423.939, E3 -213572.262}
SPL {X  -159.990, Y  +601.352, Z    +0.000, E1  +423.918, E3 -213584.048}
SPL {X  -159.990, Y  +614.998, Z    +0.000, E1  +423.962, E3 -213598.133}
SPL {X  -159.990, Y  +632.576, Z    +0.000, E1  +423.953, E3 -213616.398}
SPL {X  -159.990, Y  +648.849, Z    +0.000, E1  +423.945, E3 -213633.327}
SPL {X  -159.990, Y  +665.748, Z    +0.000, E1  +423.953, E3 -213650.883}
SPL {X  -159.643, Y  +682.032, Z    +0.000, E1  +423.894, E3 -213668.176}
SPL {X  -158.535, Y  +693.032, Z    +0.000, E1  +423.713, E3 -213680.793}
SPL {X  -156.949, Y  +702.544, Z    +0.000, E1  +423.501, E3 -213692.299}
SPL {X  -154.903, Y  +711.525, Z    +0.000, E1  +423.186, E3 -213703.770}
SPL {X  -153.138, Y  +717.820, Z    +0.000, E1  +422.909, E3 -213712.124}
SPL {X  -151.229, Y  +723.716, Z    +0.000, E1  +422.630, E3 -213720.134}
SPL {X  -149.219, Y  +729.211, Z    +0.000, E1  +422.307, E3 -213727.842}
SPL {X  -146.537, Y  +735.716, Z    +0.000, E1  +421.906, E3 -213737.185}
SPL {X  -143.476, Y  +742.291, Z    +0.000, E1  +421.379, E3 -213746.945}
SPL {X  -141.015, Y  +747.074, Z    +0.000, E1  +420.958, E3 -213754.201}
SPL {X  -138.539, Y  +751.523, Z    +0.000, E1  +420.526, E3 -213761.036}
SPL {X  -136.299, Y  +755.281, Z    +0.000, E1  +420.128, E3 -213766.897}
SPL {X  -133.306, Y  +759.967, Z    +0.000, E1  +419.584, E3 -213774.292}
SPL {X  -112.019, Y  +785.730, Z    +0.000, E1  +410.795, E3 -213877.032}
ENDSPLINE

SPLINE
SPL {X  -138.335, Y  +751.876, Z    +0.000, E1  +401.001, E3 -213991.331}
SPL {X  -150.285, Y  +726.376, Z    +0.000, E1  +392.667, E3 -214009.740}
SPL {X  -156.272, Y  +705.789, Z    +0.000, E1  +383.396, E3 -214017.377}
SPL {X  -159.413, Y  +685.076, Z    +0.000, E1  +371.341, E3 -214021.515}
SPL {X  -159.901, Y  +676.826, Z    +0.000, E1  +365.664, E3 -214022.348}
SPL {X  -159.990, Y  +671.106, Z    +0.000, E1  +361.459, E3 -214022.609}
SPL {X  -159.990, Y  +668.525, Z    +0.000, E1  +359.125, E3 -214022.655}
SPL {X  -159.990, Y  +664.817, Z    +0.000, E1  +353.836, E3 -214022.795}
SPL {X  -159.990, Y  +661.286, Z    +0.000, E1  +348.294, E3 -214023.057}
SPL {X  -159.990, Y  +656.470, Z    +0.000, E1  +340.220, E3 -214023.594}
SPL {X  -159.990, Y  +651.555, Z    +0.000, E1  +332.416, E3 -214024.402}
SPL {X  -159.990, Y  +640.109, Z    +0.000, E1  +318.471, E3 -214027.231}
SPL {X  -159.990, Y  +589.014, Z    +0.000, E1  +298.500, E3 -214049.096}
SPL {X  -159.990, Y  +484.717, Z    +0.000, E1  +295.169, E3 -214127.280}
SPL {X  -159.990, Y  +469.712, Z    +0.000, E1  +295.152, E3 -214142.217}
SPL {X  -159.990, Y  +456.089, Z    +0.000, E1  +295.174, E3 -214155.833}
SPL {X  -159.990, Y  +443.816, Z    +0.000, E1  +295.158, E3 -214168.033}
SPL {X  -159.990, Y  +405.035, Z    +0.000, E1  +292.209, E3 -214180.303}
SPL {X  -159.990, Y  +397.824, Z    +0.000, E1  +292.709, E3 -214190.665}
SPL {X  -159.990, Y  +393.786, Z    +0.000, E1  +293.391, E3 -214199.984}
SPL {X  -159.990, Y  +387.038, Z    +0.000, E1  +293.844, E3 -214209.840}
SPL {X  -159.983, Y  +380.995, Z    +0.000, E1  +294.559, E3 -214221.409}
SPL {X  -159.898, Y  +377.064, Z    +0.000, E1  +295.481, E3 -214232.223}
SPL {X  -159.533, Y  +370.414, Z    +0.000, E1  +296.253, E3 -214245.220}
SPL {X  -158.431, Y  +360.219, Z    +0.000, E1  +296.670, E3 -214258.736}
SPL {X  -157.299, Y  +353.279, Z    +0.000, E1  +296.835, E3 -214267.233}
SPL {X  -155.242, Y  +343.812, Z    +0.000, E1  +297.102, E3 -214279.281}
SPL {X  -151.999, Y  +332.569, Z    +0.000, E1  +297.592, E3 -214294.439}
SPL {X  -148.909, Y  +323.994, Z    +0.000, E1  +298.107, E3 -214306.613}
SPL {X  -146.667, Y  +318.581, Z    +0.000, E1  +298.485, E3 -214314.533}
SPL {X  -144.416, Y  +313.647, Z    +0.000, E1  +298.845, E3 -214321.869}
SPL {X  -141.484, Y  +307.808, Z    +0.000, E1  +299.342, E3 -214330.762}
SPL {X  -139.055, Y  +303.377, Z    +0.000, E1  +299.788, E3 -214337.675}
SPL {X  -136.464, Y  +298.988, Z    +0.000, E1  +300.231, E3 -214344.549}
SPL {X  -133.486, Y  +294.305, Z    +0.000, E1  +300.785, E3 -214352.011}
SPL {X  -111.268, Y  +267.538, Z    +0.000, E1  +309.436, E3 -214459.910}
ENDSPLINE

SPLINE
SPL {X  -140.331, Y  +305.662, Z    +0.000, E1  +319.927, E3 -214571.978}
SPL {X  -153.176, Y  +336.305, Z    +0.000, E1  +330.872, E3 -214590.533}
SPL {X  -157.724, Y  +355.668, Z    +0.000, E1  +340.639, E3 -214596.541}
SPL {X  -159.465, Y  +369.545, Z    +0.000, E1  +349.053, E3 -214598.863}
SPL {X  -159.983, Y  +381.031, Z    +0.000, E1  +357.053, E3 -214599.803}
SPL {X  -159.990, Y  +385.049, Z    +0.000, E1  +360.437, E3 -214599.899}
SPL {X  -159.990, Y  +389.234, Z    +0.000, E1  +366.142, E3 -214600.055}
SPL {X  -159.990, Y  +395.814, Z    +0.000, E1  +376.762, E3 -214600.656}
SPL {X  -159.990, Y  +404.858, Z    +0.000, E1  +391.125, E3 -214602.170}
SPL {X  -159.990, Y  +416.328, Z    +0.000, E1  +404.105, E3 -214605.107}
SPL {X  -159.990, Y  +459.824, Z    +0.000, E1  +420.326, E3 -214625.029}
SPL {X  -159.990, Y  +561.459, Z    +0.000, E1  +423.923, E3 -214703.896}
SPL {X  -159.990, Y  +574.787, Z    +0.000, E1  +423.950, E3 -214717.692}
SPL {X  -159.990, Y  +590.041, Z    +0.000, E1  +423.939, E3 -214733.552}
SPL {X  -159.990, Y  +601.352, Z    +0.000, E1  +423.918, E3 -214745.338}
SPL {X  -159.990, Y  +610.973, Z    +0.000, E1  +423.927, E3 -214755.306}
SPL {X  -159.990, Y  +624.756, Z    +0.000, E1  +423.949, E3 -214769.584}
SPL {X  -159.990, Y  +636.914, Z    +0.000, E1  +423.917, E3 -214782.260}
SPL {X  -159.990, Y  +648.849, Z    +0.000, E1  +423.945, E3 -214794.618}
SPL {X  -159.990, Y  +665.748, Z    +0.000, E1  +423.953, E3 -214812.173}
SPL {X  -159.643, Y  +682.032, Z    +0.000, E1  +423.894, E3 -214829.467}
SPL {X  -158.535, Y  +693.032, Z    +0.000, E1  +423.713, E3 -214842.084}
SPL {X  -156.949, Y  +702.544, Z    +0.000, E1  +423.501, E3 -214853.589}
SPL {X  -154.903, Y  +711.525, Z    +0.000, E1  +423.186, E3 -214865.060}
SPL {X  -153.138, Y  +717.820, Z    +0.000, E1  +422.909, E3 -214873.414}
SPL {X  -151.229, Y  +723.716, Z    +0.000, E1  +422.630, E3 -214881.424}
SPL {X  -148.422, Y  +731.231, Z    +0.000, E1  +422.207, E3 -214891.982}
SPL {X  -145.802, Y  +737.367, Z    +0.000, E1  +421.758, E3 -214900.935}
SPL {X  -143.476, Y  +742.291, Z    +0.000, E1  +421.379, E3 -214908.235}
SPL {X  -141.015, Y  +747.074, Z    +0.000, E1  +420.958, E3 -214915.492}
SPL {X  -137.271, Y  +753.679, Z    +0.000, E1  +420.346, E3 -214925.630}
SPL {X  -133.306, Y  +759.967, Z    +0.000, E1  +419.584, E3 -214935.582}
SPL {X  -112.019, Y  +785.730, Z    +0.000, E1  +410.795, E3 -215038.323}
ENDSPLINE

SPLINE
SPL {X  -138.335, Y  +751.876, Z    +0.000, E1  +401.001, E3 -215152.621}
SPL {X  -150.285, Y  +726.376, Z    +0.000, E1  +392.667, E3 -215171.030}
SPL {X  -154.601, Y  +712.673, Z    +0.000, E1  +386.751, E3 -215176.635}
SPL {X  -158.303, Y  +694.673, Z    +0.000, E1  +377.238, E3 -215181.304}
SPL {X  -159.774, Y  +679.819, Z    +0.000, E1  +367.840, E3 -215183.379}
SPL {X  -159.990, Y  +671.106, Z    +0.000, E1  +361.459, E3 -215183.899}
SPL {X  -159.990, Y  +668.525, Z    +0.000, E1  +359.125, E3 -215183.945}
SPL {X  -159.990, Y  +664.817, Z    +0.000, E1  +353.836, E3 -215184.085}
SPL {X  -159.990, Y  +661.286, Z    +0.000, E1  +348.294, E3 -215184.347}
SPL {X  -159.990, Y  +654.198, Z    +0.000, E1  +336.753, E3 -215185.258}
SPL {X  -159.990, Y  +643.777, Z    +0.000, E1  +322.140, E3 -215187.424}
SPL {X  -159.990, Y  +634.027, Z    +0.000, E1  +313.116, E3 -215190.335}
SPL {X  -159.990, Y  +589.014, Z    +0.000, E1  +298.500, E3 -215210.387}
SPL {X  -159.990, Y  +484.717, Z    +0.000, E1  +295.169, E3 -215288.570}
SPL {X  -159.990, Y  +469.712, Z    +0.000, E1  +295.152, E3 -215303.507}
SPL {X  -159.990, Y  +456.089, Z    +0.000, E1  +295.174, E3 -215317.123}
SPL {X  -159.990, Y  +443.816, Z    +0.000, E1  +295.158, E3 -215329.323}
SPL {X  -159.990, Y  +405.035, Z    +0.000, E1  +292.209, E3 -215341.594}
SPL {X  -159.990, Y  +397.824, Z    +0.000, E1  +292.709, E3 -215351.956}
SPL {X  -159.990, Y  +393.786, Z    +0.000, E1  +293.391, E3 -215361.275}
SPL {X  -159.990, Y  +387.038, Z    +0.000, E1  +293.844, E3 -215371.131}
SPL {X  -159.983, Y  +380.995, Z    +0.000, E1  +294.559, E3 -215382.699}
SPL {X  -159.795, Y  +374.602, Z    +0.000, E1  +295.796, E3 -215398.719}
SPL {X  -158.852, Y  +363.449, Z    +0.000, E1  +296.568, E3 -215416.092}
SPL {X  -156.653, Y  +349.995, Z    +0.000, E1  +296.892, E3 -215432.595}
SPL {X  -153.792, Y  +338.401, Z    +0.000, E1  +297.323, E3 -215447.765}
SPL {X  -151.244, Y  +330.327, Z    +0.000, E1  +297.748, E3 -215458.917}
SPL {X  -148.909, Y  +323.994, Z    +0.000, E1  +298.107, E3 -215467.903}
SPL {X  -146.667, Y  +318.581, Z    +0.000, E1  +298.485, E3 -215475.823}
SPL {X  -144.416, Y  +313.647, Z    +0.000, E1  +298.845, E3 -215483.160}
SPL {X  -141.484, Y  +307.808, Z    +0.000, E1  +299.342, E3 -215492.053}
SPL {X  -139.055, Y  +303.377, Z    +0.000, E1  +299.788, E3 -215498.965}
SPL {X  -136.464, Y  +298.988, Z    +0.000, E1  +300.231, E3 -215505.839}
SPL {X  -133.486, Y  +294.305, Z    +0.000, E1  +300.785, E3 -215513.302}
SPL {X  -111.268, Y  +267.538, Z    +0.000, E1  +309.436, E3 -215621.200}
ENDSPLINE

SPLINE
SPL {X  -140.331, Y  +305.662, Z    +0.000, E1  +319.927, E3 -215733.269}
SPL {X  -153.176, Y  +336.305, Z    +0.000, E1  +330.872, E3 -215751.823}
SPL {X  -157.724, Y  +355.668, Z    +0.000, E1  +340.639, E3 -215757.831}
SPL {X  -159.465, Y  +369.545, Z    +0.000, E1  +349.053, E3 -215760.154}
SPL {X  -159.983, Y  +381.031, Z    +0.000, E1  +357.053, E3 -215761.093}
SPL {X  -159.990, Y  +384.524, Z    +0.000, E1  +359.995, E3 -215761.181}
SPL {X  -159.990, Y  +385.853, Z    +0.000, E1  +361.539, E3 -215761.201}
SPL {X  -159.990, Y  +389.234, Z    +0.000, E1  +366.142, E3 -215761.346}
SPL {X  -159.990, Y  +395.814, Z    +0.000, E1  +376.762, E3 -215761.947}
SPL {X  -159.990, Y  +404.858, Z    +0.000, E1  +391.125, E3 -215763.460}
SPL {X  -159.990, Y  +416.328, Z    +0.000, E1  +404.105, E3 -215766.397}
SPL {X  -159.990, Y  +459.824, Z    +0.000, E1  +420.326, E3 -215786.319}
SPL {X  -159.990, Y  +561.459, Z    +0.000, E1  +423.923, E3 -215865.186}
SPL {X  -159.990, Y  +574.787, Z    +0.000, E1  +423.950, E3 -215878.982}
SPL {X  -159.990, Y  +590.041, Z    +0.000, E1  +423.939, E3 -215894.842}
SPL {X  -159.990, Y  +601.352, Z    +0.000, E1  +423.918, E3 -215906.629}
SPL {X  -159.990, Y  +614.998, Z    +0.000, E1  +423.962, E3 -215920.713}
SPL {X  -159.990, Y  +628.256, Z    +0.000, E1  +423.919, E3 -215934.562}
SPL {X  -159.990, Y  +640.674, Z    +0.000, E1  +423.943, E3 -215947.411}
SPL {X  -159.990, Y  +657.298, Z    +0.000, E1  +423.953, E3 -215964.683}
SPL {X  -159.990, Y  +670.369, Z    +0.000, E1  +423.912, E3 -215978.341}
SPL {X  -159.643, Y  +682.032, Z    +0.000, E1  +423.894, E3 -215990.757}
SPL {X  -158.535, Y  +693.032, Z    +0.000, E1  +423.713, E3 -216003.374}
SPL {X  -156.949, Y  +702.544, Z    +0.000, E1  +423.501, E3 -216014.879}
SPL {X  -154.903, Y  +711.525, Z    +0.000, E1  +423.186, E3 -216026.350}
SPL {X  -153.138, Y  +717.820, Z    +0.000, E1  +422.909, E3 -216034.705}
SPL {X  -151.229, Y  +723.716, Z    +0.000, E1  +422.630, E3 -216042.714}
SPL {X  -149.219, Y  +729.211, Z    +0.000, E1  +422.307, E3 -216050.423}
SPL {X  -146.537, Y  +735.716, Z    +0.000, E1  +421.906, E3 -216059.766}
SPL {X  -143.476, Y  +742.291, Z    +0.000, E1  +421.379, E3 -216069.526}
SPL {X  -141.015, Y  +747.074, Z    +0.000, E1  +420.958, E3 -216076.782}
SPL {X  -138.539, Y  +751.523, Z    +0.000, E1  +420.526, E3 -216083.617}
SPL {X  -136.299, Y  +755.281, Z    +0.000, E1  +420.128, E3 -216089.478}
SPL {X  -133.306, Y  +759.967, Z    +0.000, E1  +419.584, E3 -216096.872}
SPL {X  -112.019, Y  +785.730, Z    +0.000, E1  +410.795, E3 -216199.613}
ENDSPLINE

SPLINE
SPL {X  -138.335, Y  +751.876, Z    +0.000, E1  +401.001, E3 -216313.912}
SPL {X  -150.285, Y  +726.376, Z    +0.000, E1  +392.667, E3 -216332.321}
SPL {X  -154.601, Y  +712.673, Z    +0.000, E1  +386.751, E3 -216337.926}
SPL {X  -158.303, Y  +694.673, Z    +0.000, E1  +377.238, E3 -216342.595}
SPL {X  -159.774, Y  +679.819, Z    +0.000, E1  +367.840, E3 -216344.669}
SPL {X  -159.990, Y  +671.106, Z    +0.000, E1  +361.459, E3 -216345.190}
SPL {X  -159.990, Y  +669.154, Z    +0.000, E1  +359.694, E3 -216345.221}
SPL {X  -159.990, Y  +666.004, Z    +0.000, E1  +355.742, E3 -216345.321}
SPL {X  -159.990, Y  +661.286, Z    +0.000, E1  +348.294, E3 -216345.637}
SPL {X  -159.990, Y  +654.198, Z    +0.000, E1  +336.753, E3 -216346.548}
SPL {X  -159.990, Y  +640.109, Z    +0.000, E1  +318.471, E3 -216349.812}
SPL {X  -159.990, Y  +589.014, Z    +0.000, E1  +298.500, E3 -216371.677}
SPL {X  -159.990, Y  +484.717, Z    +0.000, E1  +295.169, E3 -216449.860}
SPL {X  -159.990, Y  +474.300, Z    +0.000, E1  +295.184, E3 -216460.288}
SPL {X  -159.990, Y  +465.825, Z    +0.000, E1  +295.182, E3 -216468.728}
SPL {X  -159.990, Y  +451.559, Z    +0.000, E1  +295.138, E3 -216482.864}
SPL {X  -159.990, Y  +423.512, Z    +0.000, E1  +293.559, E3 -216497.299}
SPL {X  -159.990, Y  +399.563, Z    +0.000, E1  +292.427, E3 -216509.577}
SPL {X  -159.990, Y  +393.786, Z    +0.000, E1  +293.391, E3 -216522.565}
SPL {X  -159.990, Y  +387.038, Z    +0.000, E1  +293.844, E3 -216532.421}
SPL {X  -159.983, Y  +380.995, Z    +0.000, E1  +294.559, E3 -216543.990}
SPL {X  -159.898, Y  +377.064, Z    +0.000, E1  +295.481, E3 -216554.803}
SPL {X  -159.533, Y  +370.414, Z    +0.000, E1  +296.253, E3 -216567.800}
SPL {X  -158.431, Y  +360.219, Z    +0.000, E1  +296.670, E3 -216581.317}
SPL {X  -157.299, Y  +353.279, Z    +0.000, E1  +296.835, E3 -216589.814}
SPL {X  -156.006, Y  +347.018, Z    +0.000, E1  +297.028, E3 -216597.769}
SPL {X  -153.792, Y  +338.401, Z    +0.000, E1  +297.323, E3 -216609.055}
SPL {X  -151.244, Y  +330.327, Z    +0.000, E1  +297.748, E3 -216620.208}
SPL {X  -148.909, Y  +323.994, Z    +0.000, E1  +298.107, E3 -216629.193}
SPL {X  -146.667, Y  +318.581, Z    +0.000, E1  +298.485, E3 -216637.114}
SPL {X  -144.416, Y  +313.647, Z    +0.000, E1  +298.845, E3 -216644.450}
SPL {X  -141.484, Y  +307.808, Z    +0.000, E1  +299.342, E3 -216653.343}
SPL {X  -139.055, Y  +303.377, Z    +0.000, E1  +299.788, E3 -216660.255}
SPL {X  -136.464, Y  +298.988, Z    +0.000, E1  +300.231, E3 -216667.130}
SPL {X  -133.486, Y  +294.305, Z    +0.000, E1  +300.785, E3 -216674.592}
SPL {X  -111.268, Y  +267.538, Z    +0.000, E1  +309.436, E3 -216782.491}
ENDSPLINE

SPLINE
SPL {X  -140.331, Y  +305.662, Z    +0.000, E1  +319.927, E3 -216894.559}
SPL {X  -153.176, Y  +336.305, Z    +0.000, E1  +330.872, E3 -216913.113}
SPL {X  -158.263, Y  +359.056, Z    +0.000, E1  +342.551, E3 -216919.788}
SPL {X  -159.616, Y  +371.564, Z    +0.000, E1  +350.434, E3 -216921.693}
SPL {X  -159.983, Y  +381.031, Z    +0.000, E1  +357.053, E3 -216922.383}
SPL {X  -159.990, Y  +384.524, Z    +0.000, E1  +359.995, E3 -216922.472}
SPL {X  -159.990, Y  +386.890, Z    +0.000, E1  +362.742, E3 -216922.528}
SPL {X  -159.990, Y  +392.248, Z    +0.000, E1  +370.895, E3 -216922.855}
SPL {X  -159.990, Y  +398.030, Z    +0.000, E1  +380.706, E3 -216923.506}
SPL {X  -159.990, Y  +404.858, Z    +0.000, E1  +391.125, E3 -216924.751}
SPL {X  -159.990, Y  +416.328, Z    +0.000, E1  +404.105, E3 -216927.688}
SPL {X  -159.990, Y  +459.824, Z    +0.000, E1  +420.326, E3 -216947.610}
SPL {X  -159.990, Y  +565.974, Z    +0.000, E1  +423.959, E3 -217031.098}
SPL {X  -159.990, Y  +578.588, Z    +0.000, E1  +423.918, E3 -217044.278}
SPL {X  -159.990, Y  +590.041, Z    +0.000, E1  +423.939, E3 -217056.133}
SPL {X  -159.990, Y  +601.352, Z    +0.000, E1  +423.918, E3 -217067.919}
SPL {X  -159.990, Y  +610.973, Z    +0.000, E1  +423.927, E3 -217077.887}
SPL {X  -159.990, Y  +624.756, Z    +0.000, E1  +423.949, E3 -217092.165}
SPL {X  -159.990, Y  +640.674, Z    +0.000, E1  +423.943, E3 -217108.702}
SPL {X  -159.990, Y  +652.355, Z    +0.000, E1  +423.915, E3 -217120.900}
SPL {X  -159.990, Y  +665.748, Z    +0.000, E1  +423.953, E3 -217134.754}
SPL {X  -159.643, Y  +682.032, Z    +0.000, E1  +423.894, E3 -217152.047}
SPL {X  -158.070, Y  +696.212, Z    +0.000, E1  +423.682, E3 -217168.385}
SPL {X  -155.481, Y  +709.215, Z    +0.000, E1  +423.310, E3 -217184.576}
SPL {X  -153.138, Y  +717.820, Z    +0.000, E1  +422.909, E3 -217195.995}
SPL {X  -151.229, Y  +723.716, Z    +0.000, E1  +422.630, E3 -217204.005}
SPL {X  -148.422, Y  +731.231, Z    +0.000, E1  +422.207, E3 -217214.563}
SPL {X  -145.802, Y  +737.367, Z    +0.000, E1  +421.758, E3 -217223.515}
SPL {X  -143.476, Y  +742.291, Z    +0.000, E1  +421.379, E3 -217230.816}
SPL {X  -141.015, Y  +747.074, Z    +0.000, E1  +420.958, E3 -217238.072}
SPL {X  -138.539, Y  +751.523, Z    +0.000, E1  +420.526, E3 -217244.907}
SPL {X  -136.299, Y  +755.281, Z    +0.000, E1  +420.128, E3 -217250.768}
SPL {X  -133.306, Y  +759.967, Z    +0.000, E1  +419.584, E3 -217258.163}
SPL {X  -112.019, Y  +785.730, Z    +0.000, E1  +410.795, E3 -217360.903}
ENDSPLINE

SPLINE
SPL {X  -138.335, Y  +751.876, Z    +0.000, E1  +401.001, E3 -217475.202}
SPL {X  -150.285, Y  +726.376, Z    +0.000, E1  +392.667, E3 -217493.611}
SPL {X  -154.601, Y  +712.673, Z    +0.000, E1  +386.751, E3 -217499.216}
SPL {X  -158.303, Y  +694.673, Z    +0.000, E1  +377.238, E3 -217503.885}
SPL {X  -159.774, Y  +679.819, Z    +0.000, E1  +367.840, E3 -217505.959}
SPL {X  -159.990, Y  +671.106, Z    +0.000, E1  +361.459, E3 -217506.480}
SPL {X  -159.990, Y  +669.154, Z    +0.000, E1  +359.694, E3 -217506.512}
SPL {X  -159.990, Y  +666.004, Z    +0.000, E1  +355.742, E3 -217506.611}
SPL {X  -159.990, Y  +661.286, Z    +0.000, E1  +348.294, E3 -217506.928}
SPL {X  -159.990, Y  +656.470, Z    +0.000, E1  +340.220, E3 -217507.465}
SPL {X  -159.990, Y  +651.555, Z    +0.000, E1  +332.416, E3 -217508.273}
SPL {X  -159.990, Y  +640.109, Z    +0.000, E1  +318.471, E3 -217511.102}
SPL {X  -159.990, Y  +589.014, Z    +0.000, E1  +298.500, E3 -217532.967}
SPL {X  -159.990, Y  +484.717, Z    +0.000, E1  +295.169, E3 -217611.151}
SPL {X  -159.990, Y  +474.300, Z    +0.000, E1  +295.184, E3 -217621.578}
SPL {X  -159.990, Y  +460.248, Z    +0.000, E1  +295.138, E3 -217635.488}
SPL {X  -159.990, Y  +443.816, Z    +0.000, E1  +295.158, E3 -217651.904}
SPL {X  -159.990, Y  +410.689, Z    +0.000, E1  +292.263, E3 -217659.628}
SPL {X  -159.990, Y  +399.563, Z    +0.000, E1  +292.427, E3 -217670.867}
SPL {X  -159.990, Y  +393.786, Z    +0.000, E1  +293.391, E3 -217683.855}
SPL {X  -159.990, Y  +387.038, Z    +0.000, E1  +293.844, E3 -217693.711}
SPL {X  -159.983, Y  +380.995, Z    +0.000, E1  +294.559, E3 -217705.280}
SPL {X  -159.795, Y  +374.602, Z    +0.000, E1  +295.796, E3 -217721.299}
ENDSPLINE

SPLINE
SPL {X  -159.990, Y  +389.651, Z    +0.000, E1  +300.094, E3 -217734.527}
ENDSPLINE

SPLINE
SPL {X  -159.985, Y  +381.230, Z    +0.000, E1  +300.090, E3 -217744.893}
SPL {X  -159.702, Y  +372.900, Z    +0.000, E1  +300.135, E3 -217755.430}
SPL {X  -159.030, Y  +365.001, Z    +0.000, E1  +300.230, E3 -217765.833}
SPL {X  -157.449, Y  +354.098, Z    +0.000, E1  +300.447, E3 -217780.832}
SPL {X  -155.503, Y  +344.875, Z    +0.000, E1  +300.798, E3 -217794.251}
SPL {X  -153.622, Y  +337.813, Z    +0.000, E1  +301.097, E3 -217804.844}
SPL {X  -150.877, Y  +329.275, Z    +0.000, E1  +301.527, E3 -217818.069}
SPL {X  -148.134, Y  +322.059, Z    +0.000, E1  +302.038, E3 -217829.708}
SPL {X  -145.832, Y  +316.699, Z    +0.000, E1  +302.442, E3 -217838.542}
SPL {X  -143.160, Y  +311.071, Z    +0.000, E1  +302.918, E3 -217847.987}
SPL {X  -140.427, Y  +305.839, Z    +0.000, E1  +303.430, E3 -217856.948}
SPL {X  -137.611, Y  +300.891, Z    +0.000, E1  +303.950, E3 -217865.525}
SPL {X  -121.276, Y  +278.150, Z    +0.000, E1  +311.362, E3 -217959.083}
ENDSPLINE

SPLINE
SPL {X  -121.398, Y  +278.292, Z    +0.000, E1  +311.911, E3 -217966.667}
SPL {X  -146.770, Y  +318.818, Z    +0.000, E1  +325.496, E3 -218063.704}
SPL {X  -156.430, Y  +348.936, Z    +0.000, E1  +338.153, E3 -218080.436}
SPL {X  -159.088, Y  +365.539, Z    +0.000, E1  +347.196, E3 -218084.847}
SPL {X  -159.921, Y  +377.798, Z    +0.000, E1  +354.872, E3 -218086.507}
SPL {X  -159.990, Y  +384.169, Z    +0.000, E1  +359.534, E3 -218086.862}
SPL {X  -159.990, Y  +387.385, Z    +0.000, E1  +362.811, E3 -218086.981}
SPL {X  -159.990, Y  +391.439, Z    +0.000, E1  +368.259, E3 -218087.277}
SPL {X  -159.990, Y  +395.747, Z    +0.000, E1  +374.484, E3 -218087.798}
SPL {X  -159.990, Y  +402.387, Z    +0.000, E1  +384.140, E3 -218089.031}
SPL {X  -159.990, Y  +413.408, Z    +0.000, E1  +396.965, E3 -218092.332}
SPL {X  -159.990, Y  +455.723, Z    +0.000, E1  +415.803, E3 -218114.174}
SPL {X  -159.990, Y  +537.348, Z    +0.000, E1  +420.157, E3 -218186.767}
SPL {X  -159.990, Y  +545.972, Z    +0.000, E1  +420.143, E3 -218197.301}
SPL {X  -159.990, Y  +557.131, Z    +0.000, E1  +420.184, E3 -218210.815}
SPL {X  -159.990, Y  +569.073, Z    +0.000, E1  +420.153, E3 -218225.410}
SPL {X  -159.990, Y  +577.562, Z    +0.000, E1  +420.146, E3 -218235.750}
SPL {X  -159.990, Y  +585.415, Z    +0.000, E1  +420.147, E3 -218245.315}
SPL {X  -159.990, Y  +594.125, Z    +0.000, E1  +420.153, E3 -218255.901}
SPL {X  -159.990, Y  +602.716, Z    +0.000, E1  +420.150, E3 -218266.364}
SPL {X  -159.990, Y  +612.205, Z    +0.000, E1  +420.159, E3 -218277.901}
SPL {X  -159.990, Y  +620.604, Z    +0.000, E1  +420.153, E3 -218288.116}
SPL {X  -159.990, Y  +632.106, Z    +0.000, E1  +420.183, E3 -218302.093}
SPL {X  -159.990, Y  +643.341, Z    +0.000, E1  +420.148, E3 -218315.836}
SPL {X  -159.990, Y  +652.098, Z    +0.000, E1  +420.153, E3 -218326.482}
SPL {X  -159.990, Y  +661.466, Z    +0.000, E1  +420.154, E3 -218337.893}
SPL {X  -159.963, Y  +674.441, Z    +0.000, E1  +420.189, E3 -218353.644}
SPL {X  -159.339, Y  +685.922, Z    +0.000, E1  +420.057, E3 -218368.323}
SPL {X  -158.381, Y  +694.132, Z    +0.000, E1  +419.909, E3 -218379.320}
SPL {X  -156.712, Y  +703.719, Z    +0.000, E1  +419.674, E3 -218392.685}
SPL {X  -154.922, Y  +711.450, Z    +0.000, E1  +419.348, E3 -218404.001}
SPL {X  -153.239, Y  +717.485, Z    +0.000, E1  +419.087, E3 -218413.033}
SPL {X  -150.608, Y  +725.483, Z    +0.000, E1  +418.677, E3 -218425.378}
SPL {X  -148.008, Y  +732.249, Z    +0.000, E1  +418.192, E3 -218436.245}
SPL {X  -145.943, Y  +737.055, Z    +0.000, E1  +417.829, E3 -218444.104}
SPL {X  -143.898, Y  +741.430, Z    +0.000, E1  +417.467, E3 -218451.373}
SPL {X  -141.624, Y  +745.927, Z    +0.000, E1  +417.045, E3 -218458.968}
SPL {X  -139.581, Y  +749.692, Z    +0.000, E1  +416.662, E3 -218465.415}
SPL {X  -137.120, Y  +753.931, Z    +0.000, E1  +416.213, E3 -218472.712}
SPL {X  -120.054, Y  +777.254, Z    +0.000, E1  +409.463, E3 -218559.458}
ENDSPLINE

SPLINE
SPL {X  -141.034, Y  +747.040, Z    +0.000, E1  +398.619, E3 -218667.620}
SPL {X  -152.334, Y  +720.400, Z    +0.000, E1  +389.143, E3 -218687.074}
SPL {X  -157.190, Y  +701.303, Z    +0.000, E1  +380.164, E3 -218694.235}
SPL {X  -159.460, Y  +684.516, Z    +0.000, E1  +370.556, E3 -218697.831}
SPL {X  -159.938, Y  +675.597, Z    +0.000, E1  +364.669, E3 -218698.837}
SPL {X  -159.990, Y  +669.975, Z    +0.000, E1  +360.595, E3 -218699.087}
SPL {X  -159.990, Y  +666.850, Z    +0.000, E1  +357.321, E3 -218699.188}
SPL {X  -159.990, Y  +662.495, Z    +0.000, E1  +351.318, E3 -218699.482}
SPL {X  -159.990, Y  +657.714, Z    +0.000, E1  +344.114, E3 -218700.044}
SPL {X  -159.990, Y  +651.822, Z    +0.000, E1  +335.261, E3 -218701.012}
SPL {X  -159.990, Y  +641.369, Z    +0.000, E1  +322.665, E3 -218703.850}
SPL {X  -159.990, Y  +598.251, Z    +0.000, E1  +304.104, E3 -218727.621}
SPL {X  -159.990, Y  +514.954, Z    +0.000, E1  +299.688, E3 -218801.417}
SPL {X  -159.990, Y  +505.641, Z    +0.000, E1  +299.707, E3 -218812.726}
SPL {X  -159.990, Y  +498.210, Z    +0.000, E1  +299.707, E3 -218821.719}
SPL {X  -159.990, Y  +488.988, Z    +0.000, E1  +299.693, E3 -218832.856}
SPL {X  -159.990, Y  +478.987, Z    +0.000, E1  +299.694, E3 -218844.959}
SPL {X  -159.990, Y  +468.796, Z    +0.000, E1  +299.698, E3 -218857.303}
SPL {X  -159.990, Y  +456.606, Z    +0.000, E1  +299.670, E3 -218872.008}
SPL {X  -159.990, Y  +443.890, Z    +0.000, E1  +299.691, E3 -218887.438}
SPL {X  -159.990, Y  +437.910, Z    +0.000, E1  +300.175, E3 -218897.909}
ENDSPLINE

SPLINE
SPL {X  -159.990, Y  +447.165, Z    +0.000, E1  +303.287, E3 -218906.464}
ENDSPLINE

SPLINE
SPL {X  -159.990, Y  +436.354, Z    +0.000, E1  +302.683, E3 -218917.476}
SPL {X  -159.990, Y  +425.140, Z    +0.000, E1  +301.982, E3 -218927.911}
SPL {X  -159.990, Y  +412.625, Z    +0.000, E1  +301.150, E3 -218938.747}
SPL {X  -159.990, Y  +398.951, Z    +0.000, E1  +300.353, E3 -218950.618}
SPL {X  -159.990, Y  +389.564, Z    +0.000, E1  +300.093, E3 -218960.432}
SPL {X  -159.985, Y  +381.230, Z    +0.000, E1  +300.090, E3 -218970.699}
SPL {X  -159.702, Y  +372.900, Z    +0.000, E1  +300.135, E3 -218981.236}
SPL {X  -159.030, Y  +365.001, Z    +0.000, E1  +300.230, E3 -218991.639}
SPL {X  -158.029, Y  +357.528, Z    +0.000, E1  +300.403, E3 -219001.895}
SPL {X  -156.953, Y  +351.476, Z    +0.000, E1  +300.570, E3 -219010.448}
SPL {X  -155.503, Y  +344.875, Z    +0.000, E1  +300.798, E3 -219020.057}
SPL {X  -153.622, Y  +337.813, Z    +0.000, E1  +301.097, E3 -219030.651}
SPL {X  -151.786, Y  +331.925, Z    +0.000, E1  +301.419, E3 -219039.772}
SPL {X  -150.141, Y  +327.233, Z    +0.000, E1  +301.695, E3 -219047.181}
SPL {X  -148.134, Y  +322.059, Z    +0.000, E1  +302.038, E3 -219055.514}
SPL {X  -145.832, Y  +316.699, Z    +0.000, E1  +302.442, E3 -219064.349}
SPL {X  -143.160, Y  +311.071, Z    +0.000, E1  +302.918, E3 -219073.794}
SPL {X  -140.427, Y  +305.839, Z    +0.000, E1  +303.430, E3 -219082.755}
SPL {X  -137.611, Y  +300.891, Z    +0.000, E1  +303.950, E3 -219091.331}
SPL {X  -121.335, Y  +278.219, Z    +0.000, E1  +311.699, E3 -219189.677}
ENDSPLINE

SPLINE
SPL {X  -146.770, Y  +318.818, Z    +0.000, E1  +325.496, E3 -219289.511}
SPL {X  -156.430, Y  +348.936, Z    +0.000, E1  +338.153, E3 -219306.242}
SPL {X  -159.088, Y  +365.539, Z    +0.000, E1  +347.196, E3 -219310.653}
SPL {X  -159.921, Y  +377.798, Z    +0.000, E1  +354.872, E3 -219312.313}
SPL {X  -159.990, Y  +384.169, Z    +0.000, E1  +359.534, E3 -219312.669}
SPL {X  -159.990, Y  +386.366, Z    +0.000, E1  +361.774, E3 -219312.733}
SPL {X  -159.990, Y  +390.176, Z    +0.000, E1  +366.367, E3 -219312.979}
SPL {X  -159.990, Y  +395.747, Z    +0.000, E1  +374.484, E3 -219313.605}
SPL {X  -159.990, Y  +402.387, Z    +0.000, E1  +384.140, E3 -219314.837}
SPL {X  -159.990, Y  +413.408, Z    +0.000, E1  +396.965, E3 -219318.138}
SPL {X  -159.990, Y  +455.723, Z    +0.000, E1  +415.803, E3 -219339.981}
SPL {X  -159.990, Y  +537.348, Z    +0.000, E1  +420.157, E3 -219412.573}
SPL {X  -159.990, Y  +549.907, Z    +0.000, E1  +420.183, E3 -219427.831}
SPL {X  -159.990, Y  +560.677, Z    +0.000, E1  +420.145, E3 -219441.002}
SPL {X  -159.990, Y  +569.073, Z    +0.000, E1  +420.153, E3 -219451.216}
SPL {X  -159.990, Y  +581.828, Z    +0.000, E1  +420.191, E3 -219466.675}
SPL {X  -159.990, Y  +594.125, Z    +0.000, E1  +420.153, E3 -219481.708}
SPL {X  -159.990, Y  +602.716, Z    +0.000, E1  +420.150, E3 -219492.171}
SPL {X  -159.990, Y  +612.205, Z    +0.000, E1  +420.159, E3 -219503.707}
SPL {X  -159.990, Y  +624.752, Z    +0.000, E1  +420.194, E3 -219518.915}
SPL {X  -159.990, Y  +640.062, Z    +0.000, E1  +420.188, E3 -219537.579}
SPL {X  -159.990, Y  +652.098, Z    +0.000, E1  +420.153, E3 -219552.288}
SPL {X  -159.990, Y  +661.466, Z    +0.000, E1  +420.154, E3 -219563.700}
SPL {X  -159.990, Y  +670.781, Z    +0.000, E1  +420.150, E3 -219575.047}
SPL {X  -159.839, Y  +678.445, Z    +0.000, E1  +420.123, E3 -219584.527}
SPL {X  -159.339, Y  +685.922, Z    +0.000, E1  +420.057, E3 -219594.129}
SPL {X  -158.381, Y  +694.132, Z    +0.000, E1  +419.909, E3 -219605.126}
SPL {X  -156.712, Y  +703.719, Z    +0.000, E1  +419.674, E3 -219618.491}
SPL {X  -154.922, Y  +711.450, Z    +0.000, E1  +419.348, E3 -219629.807}
SPL {X  -153.239, Y  +717.485, Z    +0.000, E1  +419.087, E3 -219638.840}
SPL {X  -150.608, Y  +725.483, Z    +0.000, E1  +418.677, E3 -219651.185}
SPL {X  -148.008, Y  +732.249, Z    +0.000, E1  +418.192, E3 -219662.051}
SPL {X  -145.943, Y  +737.055, Z    +0.000, E1  +417.829, E3 -219669.910}
SPL {X  -143.898, Y  +741.430, Z    +0.000, E1  +417.467, E3 -219677.179}
SPL {X  -141.624, Y  +745.927, Z    +0.000, E1  +417.045, E3 -219684.775}
SPL {X  -139.581, Y  +749.692, Z    +0.000, E1  +416.662, E3 -219691.221}
SPL {X  -137.120, Y  +753.931, Z    +0.000, E1  +416.213, E3 -219698.519}
SPL {X  -120.054, Y  +777.254, Z    +0.000, E1  +409.463, E3 -219785.265}
ENDSPLINE

SPLINE
SPL {X  -141.034, Y  +747.040, Z    +0.000, E1  +398.619, E3 -219893.426}
SPL {X  -152.334, Y  +720.400, Z    +0.000, E1  +389.143, E3 -219912.881}
SPL {X  -157.190, Y  +701.303, Z    +0.000, E1  +380.164, E3 -219920.041}
SPL {X  -159.460, Y  +684.516, Z    +0.000, E1  +370.556, E3 -219923.637}
SPL {X  -159.938, Y  +675.597, Z    +0.000, E1  +364.669, E3 -219924.644}
SPL {X  -159.990, Y  +671.043, Z    +0.000, E1  +361.371, E3 -219924.867}
SPL {X  -159.990, Y  +668.657, Z    +0.000, E1  +359.332, E3 -219924.928}
SPL {X  -159.990, Y  +665.812, Z    +0.000, E1  +355.875, E3 -219925.039}
SPL {X  -159.990, Y  +662.495, Z    +0.000, E1  +351.318, E3 -219925.289}
SPL {X  -159.990, Y  +657.714, Z    +0.000, E1  +344.114, E3 -219925.850}
SPL {X  -159.990, Y  +651.822, Z    +0.000, E1  +335.261, E3 -219926.818}
SPL {X  -159.990, Y  +641.369, Z    +0.000, E1  +322.665, E3 -219929.656}
SPL {X  -159.990, Y  +598.251, Z    +0.000, E1  +304.104, E3 -219953.428}
SPL {X  -159.990, Y  +514.954, Z    +0.000, E1  +299.688, E3 -220027.223}
SPL {X  -159.990, Y  +501.679, Z    +0.000, E1  +299.667, E3 -220043.260}
SPL {X  -159.990, Y  +488.988, Z    +0.000, E1  +299.693, E3 -220058.663}
SPL {X  -159.990, Y  +478.987, Z    +0.000, E1  +299.694, E3 -220070.765}
SPL {X  -159.990, Y  +468.796, Z    +0.000, E1  +299.698, E3 -220083.109}
SPL {X  -159.990, Y  +456.606, Z    +0.000, E1  +299.670, E3 -220097.815}
SPL {X  -159.990, Y  +443.890, Z    +0.000, E1  +299.691, E3 -220113.245}
SPL {X  -159.990, Y  +437.910, Z    +0.000, E1  +300.175, E3 -220123.716}
ENDSPLINE

SPLINE
SPL {X  -159.990, Y  +447.165, Z    +0.000, E1  +303.287, E3 -220132.271}
ENDSPLINE

SPLINE
SPL {X  -159.990, Y  +436.354, Z    +0.000, E1  +302.683, E3 -220143.282}
SPL {X  -159.990, Y  +425.140, Z    +0.000, E1  +301.982, E3 -220153.718}
SPL {X  -159.990, Y  +412.625, Z    +0.000, E1  +301.150, E3 -220164.554}
SPL {X  -159.990, Y  +398.951, Z    +0.000, E1  +300.353, E3 -220176.425}
SPL {X  -159.990, Y  +389.564, Z    +0.000, E1  +300.093, E3 -220186.239}
SPL {X  -159.985, Y  +381.230, Z    +0.000, E1  +300.090, E3 -220196.506}
SPL {X  -159.702, Y  +372.900, Z    +0.000, E1  +300.135, E3 -220207.043}
SPL {X  -159.030, Y  +365.001, Z    +0.000, E1  +300.230, E3 -220217.446}
SPL {X  -158.029, Y  +357.528, Z    +0.000, E1  +300.403, E3 -220227.701}
SPL {X  -156.953, Y  +351.476, Z    +0.000, E1  +300.570, E3 -220236.254}
SPL {X  -155.503, Y  +344.875, Z    +0.000, E1  +300.798, E3 -220245.864}
SPL {X  -153.622, Y  +337.813, Z    +0.000, E1  +301.097, E3 -220256.457}
SPL {X  -151.786, Y  +331.925, Z    +0.000, E1  +301.419, E3 -220265.578}
SPL {X  -150.141, Y  +327.233, Z    +0.000, E1  +301.695, E3 -220272.987}
SPL {X  -148.134, Y  +322.059, Z    +0.000, E1  +302.038, E3 -220281.321}
SPL {X  -145.832, Y  +316.699, Z    +0.000, E1  +302.442, E3 -220290.155}
SPL {X  -143.160, Y  +311.071, Z    +0.000, E1  +302.918, E3 -220299.600}
SPL {X  -140.427, Y  +305.839, Z    +0.000, E1  +303.430, E3 -220308.561}
SPL {X  -137.611, Y  +300.891, Z    +0.000, E1  +303.950, E3 -220317.137}
SPL {X  -121.335, Y  +278.219, Z    +0.000, E1  +311.699, E3 -220415.484}
ENDSPLINE

SPLINE
SPL {X  -146.770, Y  +318.818, Z    +0.000, E1  +325.496, E3 -220515.317}
SPL {X  -156.430, Y  +348.936, Z    +0.000, E1  +338.153, E3 -220532.049}
SPL {X  -159.088, Y  +365.539, Z    +0.000, E1  +347.196, E3 -220536.460}
SPL {X  -159.921, Y  +377.798, Z    +0.000, E1  +354.872, E3 -220538.120}
SPL {X  -159.990, Y  +384.169, Z    +0.000, E1  +359.534, E3 -220538.475}
SPL {X  -159.990, Y  +386.366, Z    +0.000, E1  +361.774, E3 -220538.539}
SPL {X  -159.990, Y  +390.176, Z    +0.000, E1  +366.367, E3 -220538.786}
SPL {X  -159.990, Y  +395.747, Z    +0.000, E1  +374.484, E3 -220539.411}
SPL {X  -159.990, Y  +404.190, Z    +0.000, E1  +386.444, E3 -220541.093}
SPL {X  -159.990, Y  +418.143, Z    +0.000, E1  +401.167, E3 -220545.686}
SPL {X  -159.990, Y  +460.468, Z    +0.000, E1  +416.751, E3 -220568.368}
SPL {X  -159.990, Y  +537.348, Z    +0.000, E1  +420.157, E3 -220638.380}
SPL {X  -159.990, Y  +549.907, Z    +0.000, E1  +420.183, E3 -220653.637}
SPL {X  -159.990, Y  +560.677, Z    +0.000, E1  +420.145, E3 -220666.808}
SPL {X  -159.990, Y  +569.073, Z    +0.000, E1  +420.153, E3 -220677.023}
SPL {X  -159.990, Y  +577.562, Z    +0.000, E1  +420.146, E3 -220687.362}
SPL {X  -159.990, Y  +585.415, Z    +0.000, E1  +420.147, E3 -220696.928}
SPL {X  -159.990, Y  +594.125, Z    +0.000, E1  +420.153, E3 -220707.514}
SPL {X  -159.990, Y  +602.716, Z    +0.000, E1  +420.150, E3 -220717.977}
SPL {X  -159.990, Y  +612.205, Z    +0.000, E1  +420.159, E3 -220729.514}
SPL {X  -159.990, Y  +620.604, Z    +0.000, E1  +420.153, E3 -220739.729}
SPL {X  -159.990, Y  +632.106, Z    +0.000, E1  +420.183, E3 -220753.706}
SPL {X  -159.990, Y  +643.341, Z    +0.000, E1  +420.148, E3 -220767.449}
SPL {X  -159.990, Y  +652.098, Z    +0.000, E1  +420.153, E3 -220778.095}
SPL {X  -159.990, Y  +661.466, Z    +0.000, E1  +420.154, E3 -220789.506}
SPL {X  -159.963, Y  +674.441, Z    +0.000, E1  +420.189, E3 -220805.257}
SPL {X  -159.339, Y  +685.922, Z    +0.000, E1  +420.057, E3 -220819.935}
SPL {X  -158.381, Y  +694.132, Z    +0.000, E1  +419.909, E3 -220830.933}
SPL {X  -157.192, Y  +701.291, Z    +0.000, E1  +419.715, E3 -220840.903}
SPL {X  -155.426, Y  +709.440, Z    +0.000, E1  +419.459, E3 -220852.601}
SPL {X  -153.239, Y  +717.485, Z    +0.000, E1  +419.087, E3 -220864.646}
SPL {X  -150.608, Y  +725.483, Z    +0.000, E1  +418.677, E3 -220876.991}
SPL {X  -148.008, Y  +732.249, Z    +0.000, E1  +418.192, E3 -220887.858}
SPL {X  -145.943, Y  +737.055, Z    +0.000, E1  +417.829, E3 -220895.716}
SPL {X  -143.898, Y  +741.430, Z    +0.000, E1  +417.467, E3 -220902.986}
SPL {X  -141.624, Y  +745.927, Z    +0.000, E1  +417.045, E3 -220910.581}
SPL {X  -139.581, Y  +749.692, Z    +0.000, E1  +416.662, E3 -220917.028}
SPL {X  -137.120, Y  +753.931, Z    +0.000, E1  +416.213, E3 -220924.325}
SPL {X  -120.054, Y  +777.254, Z    +0.000, E1  +409.463, E3 -221011.071}
ENDSPLINE

SPLINE
SPL {X  -141.034, Y  +747.040, Z    +0.000, E1  +398.619, E3 -221119.233}
SPL {X  -152.334, Y  +720.400, Z    +0.000, E1  +389.143, E3 -221138.687}
SPL {X  -157.190, Y  +701.303, Z    +0.000, E1  +380.164, E3 -221145.848}
SPL {X  -159.117, Y  +688.191, Z    +0.000, E1  +372.748, E3 -221148.880}
SPL {X  -159.875, Y  +677.561, Z    +0.000, E1  +366.083, E3 -221150.269}
SPL {X  -159.990, Y  +671.043, Z    +0.000, E1  +361.371, E3 -221150.673}
SPL {X  -159.990, Y  +669.269, Z    +0.000, E1  +359.855, E3 -221150.718}
SPL {X  -159.990, Y  +666.850, Z    +0.000, E1  +357.321, E3 -221150.801}
SPL {X  -159.990, Y  +662.495, Z    +0.000, E1  +351.318, E3 -221151.095}
SPL {X  -159.990, Y  +657.714, Z    +0.000, E1  +344.114, E3 -221151.656}
SPL {X  -159.990, Y  +651.822, Z    +0.000, E1  +335.261, E3 -221152.625}
SPL {X  -159.990, Y  +641.369, Z    +0.000, E1  +322.665, E3 -221155.463}
SPL {X  -159.990, Y  +598.251, Z    +0.000, E1  +304.104, E3 -221179.234}
SPL {X  -159.990, Y  +514.954, Z    +0.000, E1  +299.688, E3 -221253.030}
SPL {X  -159.990, Y  +501.679, Z    +0.000, E1  +299.667, E3 -221269.066}
SPL {X  -159.990, Y  +488.988, Z    +0.000, E1  +299.693, E3 -221284.469}
SPL {X  -159.990, Y  +478.987, Z    +0.000, E1  +299.694, E3 -221296.572}
SPL {X  -159.990, Y  +468.796, Z    +0.000, E1  +299.698, E3 -221308.915}
SPL {X  -159.990, Y  +460.399, Z    +0.000, E1  +299.707, E3 -221319.092}
SPL {X  -159.990, Y  +453.289, Z    +0.000, E1  +299.707, E3 -221327.698}
SPL {X  -159.990, Y  +443.890, Z    +0.000, E1  +299.691, E3 -221339.051}
SPL {X  -159.990, Y  +437.910, Z    +0.000, E1  +300.175, E3 -221349.522}
ENDSPLINE

SPLINE
SPL {X  -159.990, Y  +447.165, Z    +0.000, E1  +303.287, E3 -221358.077}
ENDSPLINE

SPLINE
SPL {X  -159.990, Y  +436.354, Z    +0.000, E1  +302.683, E3 -221369.089}
SPL {X  -159.990, Y  +425.140, Z    +0.000, E1  +301.982, E3 -221379.524}
SPL {X  -159.990, Y  +412.625, Z    +0.000, E1  +301.150, E3 -221390.360}
SPL {X  -159.990, Y  +398.951, Z    +0.000, E1  +300.353, E3 -221402.231}
SPL {X  -159.990, Y  +389.564, Z    +0.000, E1  +300.093, E3 -221412.045}
SPL {X  -159.985, Y  +381.230, Z    +0.000, E1  +300.090, E3 -221422.312}
SPL {X  -159.702, Y  +372.900, Z    +0.000, E1  +300.135, E3 -221432.849}
SPL {X  -159.030, Y  +365.001, Z    +0.000, E1  +300.230, E3 -221443.252}
SPL {X  -157.449, Y  +354.098, Z    +0.000, E1  +300.447, E3 -221458.252}
SPL {X  -155.503, Y  +344.875, Z    +0.000, E1  +300.798, E3 -221471.670}
SPL {X  -153.622, Y  +337.813, Z    +0.000, E1  +301.097, E3 -221482.264}
SPL {X  -150.877, Y  +329.275, Z    +0.000, E1  +301.527, E3 -221495.488}
SPL {X  -148.134, Y  +322.059, Z    +0.000, E1  +302.038, E3 -221507.127}
SPL {X  -145.832, Y  +316.699, Z    +0.000, E1  +302.442, E3 -221515.961}
SPL {X  -143.160, Y  +311.071, Z    +0.000, E1  +302.918, E3 -221525.407}
SPL {X  -140.427, Y  +305.839, Z    +0.000, E1  +303.430, E3 -221534.368}
SPL {X  -137.611, Y  +300.891, Z    +0.000, E1  +303.950, E3 -221542.944}
SPL {X  -121.335, Y  +278.219, Z    +0.000, E1  +311.699, E3 -221641.290}
ENDSPLINE

SPLINE
SPL {X  -146.770, Y  +318.818, Z    +0.000, E1  +325.496, E3 -221741.124}
SPL {X  -156.430, Y  +348.936, Z    +0.000, E1  +338.153, E3 -221757.855}
SPL {X  -159.088, Y  +365.539, Z    +0.000, E1  +347.196, E3 -221762.266}
SPL {X  -159.921, Y  +377.798, Z    +0.000, E1  +354.872, E3 -221763.926}
SPL {X  -159.990, Y  +384.169, Z    +0.000, E1  +359.534, E3 -221764.282}
SPL {X  -159.990, Y  +387.385, Z    +0.000, E1  +362.811, E3 -221764.400}
SPL {X  -159.990, Y  +391.439, Z    +0.000, E1  +368.259, E3 -221764.696}
SPL {X  -159.990, Y  +395.747, Z    +0.000, E1  +374.484, E3 -221765.217}
SPL {X  -159.990, Y  +402.387, Z    +0.000, E1  +384.140, E3 -221766.450}
SPL {X  -159.990, Y  +414.244, Z    +0.000, E1  +397.704, E3 -221770.083}
SPL {X  -159.990, Y  +460.468, Z    +0.000, E1  +416.751, E3 -221794.174}
SPL {X  -159.990, Y  +537.348, Z    +0.000, E1  +420.157, E3 -221864.186}
SPL {X  -159.990, Y  +549.907, Z    +0.000, E1  +420.183, E3 -221879.444}
SPL {X  -159.990, Y  +560.677, Z    +0.000, E1  +420.145, E3 -221892.615}
SPL {X  -159.990, Y  +569.073, Z    +0.000, E1  +420.153, E3 -221902.829}
SPL {X  -159.990, Y  +581.828, Z    +0.000, E1  +420.191, E3 -221918.288}
SPL {X  -159.990, Y  +594.125, Z    +0.000, E1  +420.153, E3 -221933.321}
SPL {X  -159.990, Y  +602.716, Z    +0.000, E1  +420.150, E3 -221943.783}
SPL {X  -159.990, Y  +612.205, Z    +0.000, E1  +420.159, E3 -221955.320}
SPL {X  -159.990, Y  +620.604, Z    +0.000, E1  +420.153, E3 -221965.536}
SPL {X  -159.990, Y  +632.106, Z    +0.000, E1  +420.183, E3 -221979.512}
SPL {X  -159.990, Y  +643.341, Z    +0.000, E1  +420.148, E3 -221993.256}
SPL {X  -159.990, Y  +652.098, Z    +0.000, E1  +420.153, E3 -222003.901}
SPL {X  -159.990, Y  +661.466, Z    +0.000, E1  +420.154, E3 -222015.312}
SPL {X  -159.963, Y  +674.441, Z    +0.000, E1  +420.189, E3 -222031.063}
SPL {X  -159.339, Y  +685.922, Z    +0.000, E1  +420.057, E3 -222045.742}
SPL {X  -158.381, Y  +694.132, Z    +0.000, E1  +419.909, E3 -222056.739}
SPL {X  -157.192, Y  +701.291, Z    +0.000, E1  +419.715, E3 -222066.710}
SPL {X  -155.426, Y  +709.440, Z    +0.000, E1  +419.459, E3 -222078.407}
SPL {X  -153.239, Y  +717.485, Z    +0.000, E1  +419.087, E3 -222090.452}
SPL {X  -150.608, Y  +725.483, Z    +0.000, E1  +418.677, E3 -222102.798}
SPL {X  -148.008, Y  +732.249, Z    +0.000, E1  +418.192, E3 -222113.664}
SPL {X  -145.943, Y  +737.055, Z    +0.000, E1  +417.829, E3 -222121.523}
SPL {X  -143.898, Y  +741.430, Z    +0.000, E1  +417.467, E3 -222128.792}
SPL {X  -141.624, Y  +745.927, Z    +0.000, E1  +417.045, E3 -222136.388}
SPL {X  -139.581, Y  +749.692, Z    +0.000, E1  +416.662, E3 -222142.834}
SPL {X  -137.120, Y  +753.931, Z    +0.000, E1  +416.213, E3 -222150.132}
SPL {X  -120.054, Y  +777.254, Z    +0.000, E1  +409.463, E3 -222236.877}
ENDSPLINE

SPLINE
SPL {X  -141.034, Y  +747.040, Z    +0.000, E1  +398.619, E3 -222345.039}
SPL {X  -152.334, Y  +720.400, Z    +0.000, E1  +389.143, E3 -222364.494}
SPL {X  -157.190, Y  +701.303, Z    +0.000, E1  +380.164, E3 -222371.654}
SPL {X  -159.117, Y  +688.191, Z    +0.000, E1  +372.748, E3 -222374.686}
SPL {X  -159.875, Y  +677.561, Z    +0.000, E1  +366.083, E3 -222376.076}
SPL {X  -159.990, Y  +669.975, Z    +0.000, E1  +360.595, E3 -222376.507}
SPL {X  -159.990, Y  +666.850, Z    +0.000, E1  +357.321, E3 -222376.607}
SPL {X  -159.990, Y  +662.495, Z    +0.000, E1  +351.318, E3 -222376.902}
SPL {X  -159.990, Y  +657.714, Z    +0.000, E1  +344.114, E3 -222377.463}
SPL {X  -159.990, Y  +651.822, Z    +0.000, E1  +335.261, E3 -222378.431}
SPL {X  -159.990, Y  +641.369, Z    +0.000, E1  +322.665, E3 -222381.269}
SPL {X  -159.990, Y  +598.251, Z    +0.000, E1  +304.104, E3 -222405.041}
SPL {X  -159.990, Y  +514.954, Z    +0.000, E1  +299.688, E3 -222478.836}
SPL {X  -159.990, Y  +505.641, Z    +0.000, E1  +299.707, E3 -222490.145}
SPL {X  -159.990, Y  +498.210, Z    +0.000, E1  +299.707, E3 -222499.139}
SPL {X  -159.990, Y  +488.988, Z    +0.000, E1  +299.693, E3 -222510.275}
SPL {X  -159.990, Y  +478.987, Z    +0.000, E1  +299.694, E3 -222522.378}
SPL {X  -159.990, Y  +468.796, Z    +0.000, E1  +299.698, E3 -222534.722}
SPL {X  -159.990, Y  +456.606, Z    +0.000, E1  +299.670, E3 -222549.428}
SPL {X  -159.990, Y  +443.890, Z    +0.000, E1  +299.691, E3 -222564.858}
SPL {X  -159.990, Y  +437.910, Z    +0.000, E1  +300.175, E3 -222575.329}
ENDSPLINE

SPLINE
SPL {X  -159.990, Y  +447.165, Z    +0.000, E1  +303.287, E3 -222583.884}
ENDSPLINE

SPLINE
SPL {X  -159.990, Y  +436.354, Z    +0.000, E1  +302.683, E3 -222594.895}
SPL {X  -159.990, Y  +425.140, Z    +0.000, E1  +301.982, E3 -222605.330}
SPL {X  -159.990, Y  +412.625, Z    +0.000, E1  +301.150, E3 -222616.167}
SPL {X  -159.990, Y  +398.951, Z    +0.000, E1  +300.353, E3 -222628.038}
SPL {X  -159.990, Y  +389.564, Z    +0.000, E1  +300.093, E3 -222637.852}
SPL {X  -159.985, Y  +381.230, Z    +0.000, E1  +300.090, E3 -222648.119}
SPL {X  -159.702, Y  +372.900, Z    +0.000, E1  +300.135, E3 -222658.656}
SPL {X  -159.030, Y  +365.001, Z    +0.000, E1  +300.230, E3 -222669.059}
SPL {X  -158.029, Y  +357.528, Z    +0.000, E1  +300.403, E3 -222679.314}
SPL {X  -156.953, Y  +351.476, Z    +0.000, E1  +300.570, E3 -222687.867}
SPL {X  -155.503, Y  +344.875, Z    +0.000, E1  +300.798, E3 -222697.477}
SPL {X  -153.622, Y  +337.813, Z    +0.000, E1  +301.097, E3 -222708.070}
SPL {X  -151.786, Y  +331.925, Z    +0.000, E1  +301.419, E3 -222717.191}
SPL {X  -150.141, Y  +327.233, Z    +0.000, E1  +301.695, E3 -222724.600}
SPL {X  -148.134, Y  +322.059, Z    +0.000, E1  +302.038, E3 -222732.934}
SPL {X  -145.832, Y  +316.699, Z    +0.000, E1  +302.442, E3 -222741.768}
SPL {X  -143.160, Y  +311.071, Z    +0.000, E1  +302.918, E3 -222751.213}
SPL {X  -140.427, Y  +305.839, Z    +0.000, E1  +303.430, E3 -222760.174}
SPL {X  -137.611, Y  +300.891, Z    +0.000, E1  +303.950, E3 -222768.750}
SPL {X  -121.335, Y  +278.219, Z    +0.000, E1  +311.699, E3 -222867.096}
ENDSPLINE

SPLINE
SPL {X  -146.770, Y  +318.818, Z    +0.000, E1  +325.496, E3 -222966.930}
SPL {X  -156.430, Y  +348.936, Z    +0.000, E1  +338.153, E3 -222983.662}
SPL {X  -159.088, Y  +365.539, Z    +0.000, E1  +347.196, E3 -222988.072}
SPL {X  -159.820, Y  +375.127, Z    +0.000, E1  +353.170, E3 -222989.496}
SPL {X  -159.990, Y  +382.134, Z    +0.000, E1  +357.935, E3 -222990.015}
SPL {X  -159.990, Y  +385.595, Z    +0.000, E1  +360.838, E3 -222990.129}
SPL {X  -159.990, Y  +390.176, Z    +0.000, E1  +366.367, E3 -222990.398}
SPL {X  -159.990, Y  +395.747, Z    +0.000, E1  +374.484, E3 -222991.024}
SPL {X  -159.990, Y  +402.387, Z    +0.000, E1  +384.140, E3 -222992.256}
SPL {X  -159.990, Y  +413.408, Z    +0.000, E1  +396.965, E3 -222995.557}
SPL {X  -159.990, Y  +455.723, Z    +0.000, E1  +415.803, E3 -223017.400}
SPL {X  -159.990, Y  +537.348, Z    +0.000, E1  +420.157, E3 -223089.992}
SPL {X  -159.990, Y  +545.972, Z    +0.000, E1  +420.143, E3 -223100.527}
SPL {X  -159.990, Y  +557.131, Z    +0.000, E1  +420.184, E3 -223114.041}
SPL {X  -159.990, Y  +569.073, Z    +0.000, E1  +420.153, E3 -223128.635}
SPL {X  -159.990, Y  +577.562, Z    +0.000, E1  +420.146, E3 -223138.975}
SPL {X  -159.990, Y  +585.415, Z    +0.000, E1  +420.147, E3 -223148.541}
SPL {X  -159.990, Y  +594.125, Z    +0.000, E1  +420.153, E3 -223159.127}
SPL {X  -159.990, Y  +602.716, Z    +0.000, E1  +420.150, E3 -223169.590}
SPL {X  -159.990, Y  +612.205, Z    +0.000, E1  +420.159, E3 -223181.126}
SPL {X  -159.990, Y  +624.752, Z    +0.000, E1  +420.194, E3 -223196.334}
SPL {X  -159.990, Y  +640.062, Z    +0.000, E1  +420.188, E3 -223214.998}
SPL {X  -159.990, Y  +652.098, Z    +0.000, E1  +420.153, E3 -223229.708}
SPL {X  -159.990, Y  +661.466, Z    +0.000, E1  +420.154, E3 -223241.119}
SPL {X  -159.963, Y  +674.441, Z    +0.000, E1  +420.189, E3 -223256.870}
SPL {X  -159.339, Y  +685.922, Z    +0.000, E1  +420.057, E3 -223271.548}
SPL {X  -158.381, Y  +694.132, Z    +0.000, E1  +419.909, E3 -223282.545}
SPL {X  -156.712, Y  +703.719, Z    +0.000, E1  +419.674, E3 -223295.910}
SPL {X  -154.922, Y  +711.450, Z    +0.000, E1  +419.348, E3 -223307.226}
SPL {X  -153.239, Y  +717.485, Z    +0.000, E1  +419.087, E3 -223316.259}
SPL {X  -150.608, Y  +725.483, Z    +0.000, E1  +418.677, E3 -223328.604}
SPL {X  -148.008, Y  +732.249, Z    +0.000, E1  +418.192, E3 -223339.471}
SPL {X  -145.943, Y  +737.055, Z    +0.000, E1  +417.829, E3 -223347.329}
SPL {X  -143.898, Y  +741.430, Z    +0.000, E1  +417.467, E3 -223354.599}
SPL {X  -140.579, Y  +747.882, Z    +0.000, E1  +416.895, E3 -223365.478}
SPL {X  -137.120, Y  +753.931, Z    +0.000, E1  +416.213, E3 -223375.938}
SPL {X  -120.054, Y  +777.254, Z    +0.000, E1  +409.463, E3 -223462.684}
ENDSPLINE

SPLINE
SPL {X  -141.034, Y  +747.040, Z    +0.000, E1  +398.619, E3 -223570.846}
SPL {X  -152.334, Y  +720.400, Z    +0.000, E1  +389.143, E3 -223590.300}
SPL {X  -157.190, Y  +701.303, Z    +0.000, E1  +380.164, E3 -223597.461}
SPL {X  -159.117, Y  +688.191, Z    +0.000, E1  +372.748, E3 -223600.493}
SPL {X  -159.875, Y  +677.561, Z    +0.000, E1  +366.083, E3 -223601.882}
SPL {X  -159.990, Y  +671.043, Z    +0.000, E1  +361.371, E3 -223602.286}
SPL {X  -159.990, Y  +669.269, Z    +0.000, E1  +359.855, E3 -223602.331}
SPL {X  -159.990, Y  +666.850, Z    +0.000, E1  +357.321, E3 -223602.414}
SPL {X  -159.990, Y  +662.495, Z    +0.000, E1  +351.318, E3 -223602.708}
SPL {X  -159.990, Y  +657.714, Z    +0.000, E1  +344.114, E3 -223603.269}
SPL {X  -159.990, Y  +651.822, Z    +0.000, E1  +335.261, E3 -223604.237}
SPL {X  -159.990, Y  +641.369, Z    +0.000, E1  +322.665, E3 -223607.076}
SPL {X  -159.990, Y  +598.251, Z    +0.000, E1  +304.104, E3 -223630.847}
SPL {X  -159.990, Y  +514.954, Z    +0.000, E1  +299.688, E3 -223704.643}
SPL {X  -159.990, Y  +501.679, Z    +0.000, E1  +299.667, E3 -223720.679}
SPL {X  -159.990, Y  +488.988, Z    +0.000, E1  +299.693, E3 -223736.082}
SPL {X  -159.990, Y  +478.987, Z    +0.000, E1  +299.694, E3 -223748.184}
SPL {X  -159.990, Y  +468.796, Z    +0.000, E1  +299.698, E3 -223760.528}
SPL {X  -159.990, Y  +456.606, Z    +0.000, E1  +299.670, E3 -223775.234}
SPL {X  -159.990, Y  +443.890, Z    +0.000, E1  +299.691, E3 -223790.664}
SPL {X  -159.990, Y  +437.910, Z    +0.000, E1  +300.175, E3 -223801.135}
ENDSPLINE

SPLINE
SPL {X  -159.990, Y  +447.165, Z    +0.000, E1  +303.287, E3 -223809.690}
ENDSPLINE

SPLINE
SPL {X  -159.990, Y  +436.354, Z    +0.000, E1  +302.683, E3 -223820.702}
SPL {X  -159.990, Y  +425.140, Z    +0.000, E1  +301.982, E3 -223831.137}
SPL {X  -159.990, Y  +412.625, Z    +0.000, E1  +301.150, E3 -223841.973}
SPL {X  -159.990, Y  +398.951, Z    +0.000, E1  +300.353, E3 -223853.844}
SPL {X  -159.990, Y  +389.564, Z    +0.000, E1  +300.093, E3 -223863.658}
SPL {X  -159.985, Y  +381.230, Z    +0.000, E1  +300.090, E3 -223873.925}
SPL {X  -159.702, Y  +372.900, Z    +0.000, E1  +300.135, E3 -223884.462}
SPL {X  -159.030, Y  +365.001, Z    +0.000, E1  +300.230, E3 -223894.865}
SPL {X  -157.449, Y  +354.098, Z    +0.000, E1  +300.447, E3 -223909.865}
SPL {X  -155.503, Y  +344.875, Z    +0.000, E1  +300.798, E3 -223923.283}
SPL {X  -153.622, Y  +337.813, Z    +0.000, E1  +301.097, E3 -223933.877}
SPL {X  -150.877, Y  +329.275, Z    +0.000, E1  +301.527, E3 -223947.101}
SPL {X  -148.134, Y  +322.059, Z    +0.000, E1  +302.038, E3 -223958.740}
SPL {X  -145.832, Y  +316.699, Z    +0.000, E1  +302.442, E3 -223967.574}
SPL {X  -143.160, Y  +311.071, Z    +0.000, E1  +302.918, E3 -223977.020}
SPL {X  -140.427, Y  +305.839, Z    +0.000, E1  +303.430, E3 -223985.981}
SPL {X  -137.611, Y  +300.891, Z    +0.000, E1  +303.950, E3 -223994.557}
SPL {X  -121.335, Y  +278.219, Z    +0.000, E1  +311.699, E3 -224092.903}
ENDSPLINE

SPLINE
SPL {X  -146.770, Y  +318.818, Z    +0.000, E1  +325.496, E3 -224192.737}
SPL {X  -156.430, Y  +348.936, Z    +0.000, E1  +338.153, E3 -224209.468}
SPL {X  -159.088, Y  +365.539, Z    +0.000, E1  +347.196, E3 -224213.879}
SPL {X  -159.921, Y  +377.798, Z    +0.000, E1  +354.872, E3 -224215.539}
SPL {X  -159.990, Y  +383.148, Z    +0.000, E1  +358.786, E3 -224215.867}
SPL {X  -159.990, Y  +385.595, Z    +0.000, E1  +360.838, E3 -224215.936}
SPL {X  -159.990, Y  +390.176, Z    +0.000, E1  +366.367, E3 -224216.205}
SPL {X  -159.990, Y  +395.747, Z    +0.000, E1  +374.484, E3 -224216.830}
SPL {X  -159.990, Y  +402.387, Z    +0.000, E1  +384.140, E3 -224218.063}
SPL {X  -159.990, Y  +413.408, Z    +0.000, E1  +396.965, E3 -224221.364}
SPL {X  -159.990, Y  +455.723, Z    +0.000, E1  +415.803, E3 -224243.206}
SPL {X  -159.990, Y  +537.348, Z    +0.000, E1  +420.157, E3 -224315.799}
SPL {X  -159.990, Y  +549.907, Z    +0.000, E1  +420.183, E3 -224331.056}
SPL {X  -159.990, Y  +560.677, Z    +0.000, E1  +420.145, E3 -224344.228}
SPL {X  -159.990, Y  +569.073, Z    +0.000, E1  +420.153, E3 -224354.442}
SPL {X  -159.990, Y  +581.828, Z    +0.000, E1  +420.191, E3 -224369.901}
SPL {X  -159.990, Y  +594.125, Z    +0.000, E1  +420.153, E3 -224384.934}
SPL {X  -159.990, Y  +602.716, Z    +0.000, E1  +420.150, E3 -224395.396}
SPL {X  -159.990, Y  +612.205, Z    +0.000, E1  +420.159, E3 -224406.933}
SPL {X  -159.990, Y  +620.604, Z    +0.000, E1  +420.153, E3 -224417.148}
SPL {X  -159.990, Y  +632.106, Z    +0.000, E1  +420.183, E3 -224431.125}
SPL {X  -159.990, Y  +643.341, Z    +0.000, E1  +420.148, E3 -224444.869}
SPL {X  -159.990, Y  +652.098, Z    +0.000, E1  +420.153, E3 -224455.514}
SPL {X  -159.990, Y  +661.466, Z    +0.000, E1  +420.154, E3 -224466.925}
SPL {X  -159.963, Y  +674.441, Z    +0.000, E1  +420.189, E3 -224482.676}
SPL {X  -159.339, Y  +685.922, Z    +0.000, E1  +420.057, E3 -224497.355}
SPL {X  -158.381, Y  +694.132, Z    +0.000, E1  +419.909, E3 -224508.352}
SPL {X  -156.712, Y  +703.719, Z    +0.000, E1  +419.674, E3 -224521.717}
SPL {X  -154.922, Y  +711.450, Z    +0.000, E1  +419.348, E3 -224533.033}
SPL {X  -153.239, Y  +717.485, Z    +0.000, E1  +419.087, E3 -224542.065}
SPL {X  -150.608, Y  +725.483, Z    +0.000, E1  +418.677, E3 -224554.411}
SPL {X  -148.008, Y  +732.249, Z    +0.000, E1  +418.192, E3 -224565.277}
SPL {X  -145.943, Y  +737.055, Z    +0.000, E1  +417.829, E3 -224573.136}
SPL {X  -143.898, Y  +741.430, Z    +0.000, E1  +417.467, E3 -224580.405}
SPL {X  -141.624, Y  +745.927, Z    +0.000, E1  +417.045, E3 -224588.000}
SPL {X  -139.581, Y  +749.692, Z    +0.000, E1  +416.662, E3 -224594.447}
SPL {X  -137.120, Y  +753.931, Z    +0.000, E1  +416.213, E3 -224601.744}
SPL {X  -120.054, Y  +777.254, Z    +0.000, E1  +409.463, E3 -224688.490}
ENDSPLINE

SPLINE
SPL {X  -141.034, Y  +747.040, Z    +0.000, E1  +398.619, E3 -224796.652}
SPL {X  -152.334, Y  +720.400, Z    +0.000, E1  +389.143, E3 -224816.107}
SPL {X  -157.190, Y  +701.303, Z    +0.000, E1  +380.164, E3 -224823.267}
SPL {X  -159.460, Y  +684.516, Z    +0.000, E1  +370.556, E3 -224826.863}
SPL {X  -159.938, Y  +675.597, Z    +0.000, E1  +364.669, E3 -224827.869}
SPL {X  -159.990, Y  +669.975, Z    +0.000, E1  +360.595, E3 -224828.120}
SPL {X  -159.990, Y  +666.850, Z    +0.000, E1  +357.321, E3 -224828.220}
SPL {X  -159.990, Y  +662.495, Z    +0.000, E1  +351.318, E3 -224828.515}
SPL {X  -159.990, Y  +657.714, Z    +0.000, E1  +344.114, E3 -224829.076}
SPL {X  -159.990, Y  +651.822, Z    +0.000, E1  +335.261, E3 -224830.044}
SPL {X  -159.990, Y  +641.369, Z    +0.000, E1  +322.665, E3 -224832.882}
SPL {X  -159.990, Y  +598.251, Z    +0.000, E1  +304.104, E3 -224856.653}
SPL {X  -159.990, Y  +514.954, Z    +0.000, E1  +299.688, E3 -224930.449}
SPL {X  -159.990, Y  +505.641, Z    +0.000, E1  +299.707, E3 -224941.758}
SPL {X  -159.990, Y  +498.210, Z    +0.000, E1  +299.707, E3 -224950.752}
SPL {X  -159.990, Y  +488.988, Z    +0.000, E1  +299.693, E3 -224961.888}
SPL {X  -159.990, Y  +478.987, Z    +0.000, E1  +299.694, E3 -224973.991}
SPL {X  -159.990, Y  +468.796, Z    +0.000, E1  +299.698, E3 -224986.335}
SPL {X  -159.990, Y  +460.399, Z    +0.000, E1  +299.707, E3 -224996.512}
SPL {X  -159.990, Y  +453.289, Z    +0.000, E1  +299.707, E3 -225005.117}
SPL {X  -159.990, Y  +443.890, Z    +0.000, E1  +299.691, E3 -225016.470}
SPL {X  -159.990, Y  +437.910, Z    +0.000, E1  +300.175, E3 -225026.941}
ENDSPLINE

SPLINE
SPL {X  -159.990, Y  +447.165, Z    +0.000, E1  +303.287, E3 -225035.497}
ENDSPLINE

SPLINE
SPL {X  -159.990, Y  +436.354, Z    +0.000, E1  +302.683, E3 -225046.508}
SPL {X  -159.990, Y  +425.140, Z    +0.000, E1  +301.982, E3 -225056.943}
SPL {X  -159.990, Y  +412.625, Z    +0.000, E1  +301.150, E3 -225067.779}
SPL {X  -159.990, Y  +398.951, Z    +0.000, E1  +300.353, E3 -225079.651}
SPL {X  -159.990, Y  +389.564, Z    +0.000, E1  +300.093, E3 -225089.465}
SPL {X  -159.985, Y  +381.230, Z    +0.000, E1  +300.090, E3 -225099.732}
SPL {X  -159.702, Y  +372.900, Z    +0.000, E1  +300.135, E3 -225110.269}
SPL {X  -159.030, Y  +365.001, Z    +0.000, E1  +300.230, E3 -225120.671}
SPL {X  -157.449, Y  +354.098, Z    +0.000, E1  +300.447, E3 -225135.671}
SPL {X  -155.503, Y  +344.875, Z    +0.000, E1  +300.798, E3 -225149.090}
SPL {X  -153.622, Y  +337.813, Z    +0.000, E1  +301.097, E3 -225159.683}
SPL {X  -150.877, Y  +329.275, Z    +0.000, E1  +301.527, E3 -225172.908}
SPL {X  -148.134, Y  +322.059, Z    +0.000, E1  +302.038, E3 -225184.546}
SPL {X  -145.832, Y  +316.699, Z    +0.000, E1  +302.442, E3 -225193.381}
SPL {X  -143.160, Y  +311.071, Z    +0.000, E1  +302.918, E3 -225202.826}
SPL {X  -140.427, Y  +305.839, Z    +0.000, E1  +303.430, E3 -225211.787}
SPL {X  -137.611, Y  +300.891, Z    +0.000, E1  +303.950, E3 -225220.363}
SPL {X  -121.335, Y  +278.219, Z    +0.000, E1  +311.699, E3 -225318.709}
ENDSPLINE

SPLINE
SPL {X  -146.770, Y  +318.818, Z    +0.000, E1  +325.496, E3 -225418.543}
SPL {X  -156.430, Y  +348.936, Z    +0.000, E1  +338.153, E3 -225435.274}
SPL {X  -159.088, Y  +365.539, Z    +0.000, E1  +347.196, E3 -225439.685}
SPL {X  -159.820, Y  +375.127, Z    +0.000, E1  +353.170, E3 -225441.109}
SPL {X  -159.990, Y  +382.134, Z    +0.000, E1  +357.935, E3 -225441.627}
SPL {X  -159.990, Y  +385.595, Z    +0.000, E1  +360.838, E3 -225441.742}
SPL {X  -159.990, Y  +390.176, Z    +0.000, E1  +366.367, E3 -225442.011}
SPL {X  -159.990, Y  +395.747, Z    +0.000, E1  +374.484, E3 -225442.637}
SPL {X  -159.990, Y  +402.387, Z    +0.000, E1  +384.140, E3 -225443.869}
SPL {X  -159.990, Y  +414.244, Z    +0.000, E1  +397.704, E3 -225447.502}
SPL {X  -159.990, Y  +460.468, Z    +0.000, E1  +416.751, E3 -225471.594}
SPL {X  -159.990, Y  +537.348, Z    +0.000, E1  +420.157, E3 -225541.605}
SPL {X  -159.990, Y  +545.972, Z    +0.000, E1  +420.143, E3 -225552.139}
SPL {X  -159.990, Y  +557.131, Z    +0.000, E1  +420.184, E3 -225565.654}
SPL {X  -159.990, Y  +569.073, Z    +0.000, E1  +420.153, E3 -225580.248}
SPL {X  -159.990, Y  +577.562, Z    +0.000, E1  +420.146, E3 -225590.588}
SPL {X  -159.990, Y  +585.415, Z    +0.000, E1  +420.147, E3 -225600.154}
SPL {X  -159.990, Y  +594.125, Z    +0.000, E1  +420.153, E3 -225610.740}
SPL {X  -159.990, Y  +602.716, Z    +0.000, E1  +420.150, E3 -225621.203}
SPL {X  -159.990, Y  +612.205, Z    +0.000, E1  +420.159, E3 -225632.739}
SPL {X  -159.990, Y  +624.752, Z    +0.000, E1  +420.194, E3 -225647.947}
SPL {X  -159.990, Y  +640.062, Z    +0.000, E1  +420.188, E3 -225666.611}
SPL {X  -159.990, Y  +652.098, Z    +0.000, E1  +420.153, E3 -225681.320}
SPL {X  -159.990, Y  +661.466, Z    +0.000, E1  +420.154, E3 -225692.732}
SPL {X  -159.963, Y  +674.441, Z    +0.000, E1  +420.189, E3 -225708.482}
SPL {X  -159.339, Y  +685.922, Z    +0.000, E1  +420.057, E3 -225723.161}
SPL {X  -158.381, Y  +694.132, Z    +0.000, E1  +419.909, E3 -225734.158}
SPL {X  -157.192, Y  +701.291, Z    +0.000, E1  +419.715, E3 -225744.129}
SPL {X  -155.426, Y  +709.440, Z    +0.000, E1  +419.459, E3 -225755.827}
SPL {X  -153.239, Y  +717.485, Z    +0.000, E1  +419.087, E3 -225767.872}
SPL {X  -150.608, Y  +725.483, Z    +0.000, E1  +418.677, E3 -225780.217}
SPL {X  -148.008, Y  +732.249, Z    +0.000, E1  +418.192, E3 -225791.084}
SPL {X  -145.943, Y  +737.055, Z    +0.000, E1  +417.829, E3 -225798.942}
SPL {X  -143.898, Y  +741.430, Z    +0.000, E1  +417.467, E3 -225806.212}
SPL {X  -140.579, Y  +747.882, Z    +0.000, E1  +416.895, E3 -225817.091}
SPL {X  -137.120, Y  +753.931, Z    +0.000, E1  +416.213, E3 -225827.551}
SPL {X  -120.054, Y  +777.254, Z    +0.000, E1  +409.463, E3 -225914.297}
ENDSPLINE

SPLINE
SPL {X  -141.034, Y  +747.040, Z    +0.000, E1  +398.619, E3 -226022.459}
SPL {X  -152.334, Y  +720.400, Z    +0.000, E1  +389.143, E3 -226041.913}
SPL {X  -157.190, Y  +701.303, Z    +0.000, E1  +380.164, E3 -226049.074}
SPL {X  -159.117, Y  +688.191, Z    +0.000, E1  +372.748, E3 -226052.106}
SPL {X  -159.875, Y  +677.561, Z    +0.000, E1  +366.083, E3 -226053.495}
SPL {X  -159.990, Y  +671.043, Z    +0.000, E1  +361.371, E3 -226053.899}
SPL {X  -159.990, Y  +669.269, Z    +0.000, E1  +359.855, E3 -226053.944}
SPL {X  -159.990, Y  +666.850, Z    +0.000, E1  +357.321, E3 -226054.026}
SPL {X  -159.990, Y  +662.495, Z    +0.000, E1  +351.318, E3 -226054.321}
SPL {X  -159.990, Y  +657.714, Z    +0.000, E1  +344.114, E3 -226054.882}
SPL {X  -159.990, Y  +651.822, Z    +0.000, E1  +335.261, E3 -226055.850}
SPL {X  -159.990, Y  +641.369, Z    +0.000, E1  +322.665, E3 -226058.689}
SPL {X  -159.990, Y  +598.251, Z    +0.000, E1  +304.104, E3 -226082.460}
SPL {X  -159.990, Y  +514.954, Z    +0.000, E1  +299.688, E3 -226156.255}
SPL {X  -159.990, Y  +505.641, Z    +0.000, E1  +299.707, E3 -226167.564}
SPL {X  -159.990, Y  +498.210, Z    +0.000, E1  +299.707, E3 -226176.558}
SPL {X  -159.990, Y  +488.988, Z    +0.000, E1  +299.693, E3 -226187.695}
SPL {X  -159.990, Y  +478.987, Z    +0.000, E1  +299.694, E3 -226199.797}
SPL {X  -159.990, Y  +468.796, Z    +0.000, E1  +299.698, E3 -226212.141}
SPL {X  -159.990, Y  +460.399, Z    +0.000, E1  +299.707, E3 -226222.318}
SPL {X  -159.990, Y  +453.289, Z    +0.000, E1  +299.707, E3 -226230.924}
SPL {X  -159.990, Y  +443.890, Z    +0.000, E1  +299.691, E3 -226242.277}
SPL {X  -159.990, Y  +437.910, Z    +0.000, E1  +300.175, E3 -226252.748}
ENDSPLINE

SPLINE
SPL {X  -159.990, Y  +447.165, Z    +0.000, E1  +303.287, E3 -226261.303}
ENDSPLINE

SPLINE
SPL {X  -159.990, Y  +436.354, Z    +0.000, E1  +302.683, E3 -226272.314}
SPL {X  -159.990, Y  +425.140, Z    +0.000, E1  +301.982, E3 -226282.750}
SPL {X  -159.990, Y  +412.625, Z    +0.000, E1  +301.150, E3 -226293.586}
SPL {X  -159.990, Y  +398.951, Z    +0.000, E1  +300.353, E3 -226305.457}
SPL {X  -159.990, Y  +389.564, Z    +0.000, E1  +300.093, E3 -226315.271}
SPL {X  -159.985, Y  +381.230, Z    +0.000, E1  +300.090, E3 -226325.538}
SPL {X  -159.702, Y  +372.900, Z    +0.000, E1  +300.135, E3 -226336.075}
SPL {X  -159.030, Y  +365.001, Z    +0.000, E1  +300.230, E3 -226346.478}
SPL {X  -158.029, Y  +357.528, Z    +0.000, E1  +300.403, E3 -226356.733}
SPL {X  -156.953, Y  +351.476, Z    +0.000, E1  +300.570, E3 -226365.287}
SPL {X  -155.503, Y  +344.875, Z    +0.000, E1  +300.798, E3 -226374.896}
SPL {X  -153.622, Y  +337.813, Z    +0.000, E1  +301.097, E3 -226385.490}
SPL {X  -151.786, Y  +331.925, Z    +0.000, E1  +301.419, E3 -226394.610}
SPL {X  -150.141, Y  +327.233, Z    +0.000, E1  +301.695, E3 -226402.019}
SPL {X  -148.134, Y  +322.059, Z    +0.000, E1  +302.038, E3 -226410.353}
SPL {X  -145.832, Y  +316.699, Z    +0.000, E1  +302.442, E3 -226419.187}
SPL {X  -143.160, Y  +311.071, Z    +0.000, E1  +302.918, E3 -226428.632}
SPL {X  -140.427, Y  +305.839, Z    +0.000, E1  +303.430, E3 -226437.594}
SPL {X  -137.611, Y  +300.891, Z    +0.000, E1  +303.950, E3 -226446.170}
SPL {X  -121.335, Y  +278.219, Z    +0.000, E1  +311.699, E3 -226544.516}
ENDSPLINE

SPLINE
SPL {X  -146.770, Y  +318.818, Z    +0.000, E1  +325.496, E3 -226644.350}
SPL {X  -156.430, Y  +348.936, Z    +0.000, E1  +338.153, E3 -226661.081}
SPL {X  -159.088, Y  +365.539, Z    +0.000, E1  +347.196, E3 -226665.492}
SPL {X  -159.921, Y  +377.798, Z    +0.000, E1  +354.872, E3 -226667.152}
SPL {X  -159.990, Y  +383.148, Z    +0.000, E1  +358.786, E3 -226667.479}
SPL {X  -159.990, Y  +384.761, Z    +0.000, E1  +360.138, E3 -226667.524}
SPL {X  -159.990, Y  +387.385, Z    +0.000, E1  +362.811, E3 -226667.626}
SPL {X  -159.990, Y  +391.439, Z    +0.000, E1  +368.259, E3 -226667.922}
SPL {X  -159.990, Y  +395.747, Z    +0.000, E1  +374.484, E3 -226668.443}
SPL {X  -159.990, Y  +402.387, Z    +0.000, E1  +384.140, E3 -226669.676}
SPL {X  -159.990, Y  +414.244, Z    +0.000, E1  +397.704, E3 -226673.309}
SPL {X  -159.990, Y  +460.468, Z    +0.000, E1  +416.751, E3 -226697.400}
SPL {X  -159.990, Y  +537.348, Z    +0.000, E1  +420.157, E3 -226767.412}
SPL {X  -159.990, Y  +549.907, Z    +0.000, E1  +420.183, E3 -226782.669}
SPL {X  -159.990, Y  +560.677, Z    +0.000, E1  +420.145, E3 -226795.840}
SPL {X  -159.990, Y  +569.073, Z    +0.000, E1  +420.153, E3 -226806.055}
SPL {X  -159.990, Y  +577.562, Z    +0.000, E1  +420.146, E3 -226816.395}
SPL {X  -159.990, Y  +585.415, Z    +0.000, E1  +420.147, E3 -226825.960}
SPL {X  -159.990, Y  +594.125, Z    +0.000, E1  +420.153, E3 -226836.547}
SPL {X  -159.990, Y  +602.716, Z    +0.000, E1  +420.150, E3 -226847.009}
SPL {X  -159.990, Y  +612.205, Z    +0.000, E1  +420.159, E3 -226858.546}
SPL {X  -159.990, Y  +620.604, Z    +0.000, E1  +420.153, E3 -226868.761}
SPL {X  -159.990, Y  +632.106, Z    +0.000, E1  +420.183, E3 -226882.738}
SPL {X  -159.990, Y  +643.341, Z    +0.000, E1  +420.148, E3 -226896.482}
SPL {X  -159.990, Y  +652.098, Z    +0.000, E1  +420.153, E3 -226907.127}
SPL {X  -159.990, Y  +661.466, Z    +0.000, E1  +420.154, E3 -226918.538}
SPL {X  -159.990, Y  +670.781, Z    +0.000, E1  +420.150, E3 -226929.886}
SPL {X  -159.839, Y  +678.445, Z    +0.000, E1  +420.123, E3 -226939.365}
SPL {X  -159.339, Y  +685.922, Z    +0.000, E1  +420.057, E3 -226948.968}
SPL {X  -158.381, Y  +694.132, Z    +0.000, E1  +419.909, E3 -226959.965}
SPL {X  -157.192, Y  +701.291, Z    +0.000, E1  +419.715, E3 -226969.935}
SPL {X  -155.426, Y  +709.440, Z    +0.000, E1  +419.459, E3 -226981.633}
SPL {X  -153.239, Y  +717.485, Z    +0.000, E1  +419.087, E3 -226993.678}
SPL {X  -151.467, Y  +723.022, Z    +0.000, E1  +418.780, E3 -227002.230}
SPL {X  -148.791, Y  +730.306, Z    +0.000, E1  +418.370, E3 -227013.695}
SPL {X  -145.943, Y  +737.055, Z    +0.000, E1  +417.829, E3 -227024.749}
SPL {X  -143.898, Y  +741.430, Z    +0.000, E1  +417.467, E3 -227032.018}
SPL {X  -141.624, Y  +745.927, Z    +0.000, E1  +417.045, E3 -227039.613}
SPL {X  -139.581, Y  +749.692, Z    +0.000, E1  +416.662, E3 -227046.060}
SPL {X  -137.120, Y  +753.931, Z    +0.000, E1  +416.213, E3 -227053.357}
SPL {X  -120.054, Y  +777.254, Z    +0.000, E1  +409.463, E3 -227140.103}
ENDSPLINE

